LIN {X 0,Y 409.894,Z 382.469,A -85,B 0,C 180,E1 -10359.873,E2 -10359.873} C_VEL
LIN {X 0,Y 410.199,Z 379.368,A -85,B 0,C 180,E1 -10361.865,E2 -10361.865} C_VEL
LIN {X 0,Y 410.49,Z 374.761,A -85,B 0,C 180,E1 -10363.869,E2 -10363.869} C_VEL
LIN {X 0,Y 410.864,Z 370.201,A -85,B 0,C 180,E1 -10365.375,E2 -10365.375} C_VEL
LIN {X 0,Y 411.455,Z 364.311,A -85,B 0,C 180,E1 -10366.955,E2 -10366.955} C_VEL
LIN {X 0,Y 412.195,Z 356.607,A -85,B 0,C 180,E1 -10368.644,E2 -10368.644} C_VEL
LIN {X 0,Y 413.203,Z 347.062,A -85,B 0,C 180,E1 -10370.341,E2 -10370.341} C_VEL
LIN {X 0,Y 414.197,Z 338.033,A -85,B 0,C 180,E1 -10371.657,E2 -10371.657} C_VEL
LIN {X 0,Y 415.184,Z 327.747,A -85,B 0,C 180,E1 -10372.913,E2 -10372.913} C_VEL
LIN {X 0,Y 416.321,Z 316.334,A -85,B 0,C 180,E1 -10374.056,E2 -10374.056} C_VEL
LIN {X 0,Y 417.327,Z 304.389,A -85,B 0,C 180,E1 -10375.032,E2 -10375.032} C_VEL
LIN {X 0,Y 418.436,Z 290.839,A -85,B 0,C 180,E1 -10375.893,E2 -10375.893} C_VEL
LIN {X 0,Y 419.174,Z 276.579,A -85,B 0,C 180,E1 -10376.58,E2 -10376.58} C_VEL
LIN {X 0,Y 419.797,Z 262.212,A -85,B 0,C 180,E1 -10377.052,E2 -10377.052} C_VEL
LIN {X 0,Y 420.231,Z 239.052,A -85,B 0,C 180,E1 -10377.499,E2 -10377.499} C_VEL
LIN {X 0,Y 421.741,Z 148.538,A -85,B 0,C 180,E1 -10379.069,E2 -10379.069} C_VEL
LIN {X 0,Y 417.255,Z 129.702,A -85,B 0,C 180,E1 -10379.713,E2 -10379.713} C_VEL
LIN {X 0,Y 414.712,Z 123.273,A -85,B 0,C 180,E1 -10380.021,E2 -10380.021} C_VEL
LIN {X 0,Y 411.925,Z 110.451,A -85,B 0,C 180,E1 -10383.091,E2 -10383.091} C_VEL
LIN {X 0,Y 411.225,Z 107.391,A -85,B 0,C 180,E1 -10383.888,E2 -10383.888} C_VEL
LIN {X 0,Y 411.186,Z 107.387,A -85,B 0,C 180,E1 -10386.743,E2 -10386.743} C_VEL
LIN {X 0,Y 411.164,Z 107.396,A -85,B 0,C 180,E1 -10389.719,E2 -10389.719} C_VEL
LIN {X 0,Y 411.162,Z 107.393,A -85,B 0,C 180,E1 -10393.135,E2 -10393.135} C_VEL
LIN {X 0,Y 411.164,Z 107.386,A -85,B 0,C 180,E1 -10395.882,E2 -10395.882} C_VEL
LIN {X 0,Y 411.148,Z 107.394,A -85,B 0,C 180,E1 -10398.774,E2 -10398.774} C_VEL
LIN {X 0,Y 411.183,Z 107.39,A -85,B 0,C 180,E1 -10402.025,E2 -10402.025} C_VEL
LIN {X 0,Y 411.203,Z 107.389,A -85,B 0,C 180,E1 -10405.123,E2 -10405.123} C_VEL
LIN {X 0,Y 411.166,Z 107.391,A -85,B 0,C 180,E1 -10408.002,E2 -10408.002} C_VEL
LIN {X 0,Y 411.181,Z 107.392,A -85,B 0,C 180,E1 -10411.407,E2 -10411.407} C_VEL
LIN {X 0,Y 411.213,Z 107.388,A -85,B 0,C 180,E1 -10414.934,E2 -10414.934} C_VEL
LIN {X 0,Y 411.204,Z 107.38,A -85,B 0,C 180,E1 -10417.913,E2 -10417.913} C_VEL
LIN {X 0,Y 411.22,Z 107.381,A -85,B 0,C 180,E1 -10421.051,E2 -10421.051} C_VEL
LIN {X 0,Y 411.254,Z 107.382,A -85,B 0,C 180,E1 -10424.131,E2 -10424.131} C_VEL
LIN {X 0,Y 411.304,Z 107.371,A -85,B 0,C 180,E1 -10427.165,E2 -10427.165} C_VEL
LIN {X 0,Y 411.292,Z 107.375,A -85,B 0,C 180,E1 -10430.161,E2 -10430.161} C_VEL
LIN {X 0,Y 411.424,Z 107.358,A -85,B 0,C 180,E1 -10433.132,E2 -10433.132} C_VEL
LIN {X 0,Y 411.304,Z 107.371,A -85,B 0,C 180,E1 -10435.099,E2 -10435.099} C_VEL
LIN {X 0,Y 411.511,Z 107.351,A -85,B 0,C 180,E1 -10438.042,E2 -10438.042} C_VEL
LIN {X 0,Y 411.639,Z 107.332,A -85,B 0,C 180,E1 -10440,E2 -10440} C_VEL
LIN {X 0,Y 411.451,Z 107.354,A -85,B 0,C 180,E1 -10442.937,E2 -10442.937} C_VEL
LIN {X 0,Y 411.435,Z 107.353,A -85,B 0,C 180,E1 -10445.882,E2 -10445.882} C_VEL
LIN {X 0,Y 411.319,Z 107.372,A -85,B 0,C 180,E1 -10448.846,E2 -10448.846} C_VEL
LIN {X 0,Y 411.284,Z 107.374,A -85,B 0,C 180,E1 -10451.833,E2 -10451.833} C_VEL
LIN {X 0,Y 411.26,Z 107.38,A -85,B 0,C 180,E1 -10454.853,E2 -10454.853} C_VEL
LIN {X 0,Y 411.253,Z 107.38,A -85,B 0,C 180,E1 -10457.915,E2 -10457.915} C_VEL
LIN {X 0,Y 411.197,Z 107.383,A -85,B 0,C 180,E1 -10461.034,E2 -10461.034} C_VEL
LIN {X 0,Y 411.228,Z 107.38,A -85,B 0,C 180,E1 -10464.215,E2 -10464.215} C_VEL
LIN {X 0,Y 411.259,Z 107.378,A -85,B 0,C 180,E1 -10467.478,E2 -10467.478} C_VEL
LIN {X 0,Y 411.19,Z 107.392,A -85,B 0,C 180,E1 -10470.847,E2 -10470.847} C_VEL
LIN {X 0,Y 411.207,Z 107.389,A -85,B 0,C 180,E1 -10474.333,E2 -10474.333} C_VEL
LIN {X 0,Y 411.192,Z 107.389,A -85,B 0,C 180,E1 -10477.974,E2 -10477.974} C_VEL
LIN {X 0,Y 411.164,Z 107.39,A -85,B 0,C 180,E1 -10481.228,E2 -10481.228} C_VEL
LIN {X 0,Y 411.176,Z 107.383,A -85,B 0,C 180,E1 -10484.49,E2 -10484.49} C_VEL
LIN {X 0,Y 411.178,Z 107.394,A -85,B 0,C 180,E1 -10488.195,E2 -10488.195} C_VEL
LIN {X 0,Y 411.223,Z 107.382,A -85,B 0,C 180,E1 -10490.776,E2 -10490.776} C_VEL
LIN {X 0,Y 411.199,Z 107.386,A -85,B 0,C 180,E1 -10494.471,E2 -10494.471} C_VEL
LIN {X 0,Y 411.208,Z 107.379,A -85,B 0,C 180,E1 -10496.873,E2 -10496.873} C_VEL
LIN {X 0,Y 411.225,Z 107.421,A -85,B 0,C 180,E1 -10499.227,E2 -10499.227} C_VEL
LIN {X 0,Y 414.619,Z 121.415,A -85,B 0,C 180,E1 -10502.366,E2 -10502.366} C_VEL
LIN {X 0,Y 416.242,Z 130.214,A -85,B 0,C 180,E1 -10504.229,E2 -10504.229} C_VEL
LIN {X 0,Y 415.402,Z 139.95,A -85,B 0,C 180,E1 -10506.075,E2 -10506.075} C_VEL
LIN {X 0,Y 421.021,Z 167.755,A -85,B 0,C 180,E1 -10506.967,E2 -10506.967} C_VEL
LIN {X 0,Y 421.464,Z 172.933,A -85,B 0,C 180,E1 -10507.09,E2 -10507.09} C_VEL
LIN {X 0,Y 419.669,Z 277.802,A -85,B 0,C 180,E1 -10508.929,E2 -10508.929} C_VEL
LIN {X 0,Y 418.967,Z 292.415,A -85,B 0,C 180,E1 -10509.374,E2 -10509.374} C_VEL
LIN {X 0,Y 418.091,Z 305.794,A -85,B 0,C 180,E1 -10509.971,E2 -10509.971} C_VEL
LIN {X 0,Y 417.093,Z 319.845,A -85,B 0,C 180,E1 -10510.825,E2 -10510.825} C_VEL
LIN {X 0,Y 416.008,Z 332.243,A -85,B 0,C 180,E1 -10511.788,E2 -10511.788} C_VEL
LIN {X 0,Y 414.859,Z 343.663,A -85,B 0,C 180,E1 -10512.882,E2 -10512.882} C_VEL
LIN {X 0,Y 413.673,Z 355.136,A -85,B 0,C 180,E1 -10514.227,E2 -10514.227} C_VEL
LIN {X 0,Y 412.634,Z 365.412,A -85,B 0,C 180,E1 -10515.702,E2 -10515.702} C_VEL
LIN {X 0,Y 411.827,Z 373.917,A -85,B 0,C 180,E1 -10517.182,E2 -10517.182} C_VEL
LIN {X 0,Y 411.039,Z 382.063,A -85,B 0,C 180,E1 -10518.91,E2 -10518.91} C_VEL
LIN {X 0,Y 410.52,Z 388.644,A -85,B 0,C 180,E1 -10520.64,E2 -10520.64} C_VEL
LIN {X 0,Y 410.161,Z 394.498,A -85,B 0,C 180,E1 -10522.616,E2 -10522.616} C_VEL
LIN {X 0,Y 409.998,Z 397.888,A -85,B 0,C 180,E1 -10524.097,E2 -10524.097} C_VEL
LIN {X 0,Y 409.904,Z 401.081,A -85,B 0,C 180,E1 -10526.067,E2 -10526.067} C_VEL
LIN {X 0,Y 409.958,Z 402.906,A -85,B 0,C 180,E1 -10528.035,E2 -10528.035} C_VEL
LIN {X 0,Y 409.905,Z 403.396,A -85,B 0,C 180,E1 -10530,E2 -10530} C_VEL
LIN {X 0,Y 409.963,Z 402.557,A -85,B 0,C 180,E1 -10531.965,E2 -10531.965} C_VEL
LIN {X 0,Y 409.904,Z 400.363,A -85,B 0,C 180,E1 -10533.932,E2 -10533.932} C_VEL
LIN {X 0,Y 409.976,Z 396.757,A -85,B 0,C 180,E1 -10535.903,E2 -10535.903} C_VEL
LIN {X 0,Y 410.181,Z 391.629,A -85,B 0,C 180,E1 -10537.878,E2 -10537.878} C_VEL
LIN {X 0,Y 410.447,Z 386.655,A -85,B 0,C 180,E1 -10539.362,E2 -10539.362} C_VEL
LIN {X 0,Y 410.935,Z 379.509,A -85,B 0,C 180,E1 -10541.093,E2 -10541.093} C_VEL
LIN {X 0,Y 411.493,Z 372.023,A -85,B 0,C 180,E1 -10542.577,E2 -10542.577} C_VEL
LIN {X 0,Y 412.153,Z 363.017,A -85,B 0,C 180,E1 -10544.063,E2 -10544.063} C_VEL
LIN {X 0,Y 412.956,Z 354.075,A -85,B 0,C 180,E1 -10545.295,E2 -10545.295} C_VEL
LIN {X 0,Y 413.778,Z 343.393,A -85,B 0,C 180,E1 -10546.529,E2 -10546.529} C_VEL
LIN {X 0,Y 414.78,Z 331.746,A -85,B 0,C 180,E1 -10547.63,E2 -10547.63} C_VEL
LIN {X 0,Y 415.787,Z 318.934,A -85,B 0,C 180,E1 -10548.605,E2 -10548.605} C_VEL
LIN {X 0,Y 416.63,Z 305.594,A -85,B 0,C 180,E1 -10549.399,E2 -10549.399} C_VEL
LIN {X 0,Y 417.339,Z 291.973,A -85,B 0,C 180,E1 -10550.002,E2 -10550.002} C_VEL
LIN {X 0,Y 417.882,Z 278.039,A -85,B 0,C 180,E1 -10550.425,E2 -10550.425} C_VEL
LIN {X 0,Y 419.494,Z 169.965,A -85,B 0,C 180,E1 -10552.298,E2 -10552.298} C_VEL
LIN {X 0,Y 414.351,Z 140.071,A -85,B 0,C 180,E1 -10553.116,E2 -10553.116} C_VEL
LIN {X 0,Y 415.279,Z 126.829,A -85,B 0,C 180,E1 -10555.566,E2 -10555.566} C_VEL
LIN {X 0,Y 413.122,Z 115.869,A -85,B 0,C 180,E1 -10557.795,E2 -10557.795} C_VEL
LIN {X 0,Y 411.225,Z 107.388,A -85,B 0,C 180,E1 -10559.597,E2 -10559.597} C_VEL
LIN {X 0,Y 411.206,Z 107.385,A -85,B 0,C 180,E1 -10563.156,E2 -10563.156} C_VEL
LIN {X 0,Y 411.192,Z 107.388,A -85,B 0,C 180,E1 -10566.552,E2 -10566.552} C_VEL
LIN {X 0,Y 411.212,Z 107.388,A -85,B 0,C 180,E1 -10569.728,E2 -10569.728} C_VEL
LIN {X 0,Y 411.174,Z 107.389,A -85,B 0,C 180,E1 -10573.133,E2 -10573.133} C_VEL
LIN {X 0,Y 411.233,Z 107.387,A -85,B 0,C 180,E1 -10575.871,E2 -10575.871} C_VEL
LIN {X 0,Y 411.204,Z 107.385,A -85,B 0,C 180,E1 -10578.765,E2 -10578.765} C_VEL
LIN {X 0,Y 411.19,Z 107.389,A -85,B 0,C 180,E1 -10582.026,E2 -10582.026} C_VEL
LIN {X 0,Y 411.204,Z 107.389,A -85,B 0,C 180,E1 -10585.666,E2 -10585.666} C_VEL
LIN {X 0,Y 411.188,Z 107.392,A -85,B 0,C 180,E1 -10589.152,E2 -10589.152} C_VEL
LIN {X 0,Y 411.257,Z 107.379,A -85,B 0,C 180,E1 -10592.522,E2 -10592.522} C_VEL
LIN {X 0,Y 411.225,Z 107.383,A -85,B 0,C 180,E1 -10595.785,E2 -10595.785} C_VEL
LIN {X 0,Y 411.195,Z 107.393,A -85,B 0,C 180,E1 -10598.966,E2 -10598.966} C_VEL
LIN {X 0,Y 411.251,Z 107.379,A -85,B 0,C 180,E1 -10602.085,E2 -10602.085} C_VEL
LIN {X 0,Y 411.259,Z 107.381,A -85,B 0,C 180,E1 -10605.147,E2 -10605.147} C_VEL
LIN {X 0,Y 411.283,Z 107.377,A -85,B 0,C 180,E1 -10608.167,E2 -10608.167} C_VEL
LIN {X 0,Y 411.439,Z 107.358,A -85,B 0,C 180,E1 -10612.189,E2 -10612.189} C_VEL
LIN {X 0,Y 411.471,Z 107.354,A -85,B 0,C 180,E1 -10614.118,E2 -10614.118} C_VEL
LIN {X 0,Y 411.51,Z 107.35,A -85,B 0,C 180,E1 -10618.043,E2 -10618.043} C_VEL
LIN {X 0,Y 411.639,Z 107.334,A -85,B 0,C 180,E1 -10620,E2 -10620} C_VEL
LIN {X 0,Y 411.457,Z 107.354,A -85,B 0,C 180,E1 -10622.937,E2 -10622.937} C_VEL
LIN {X 0,Y 411.421,Z 107.358,A -85,B 0,C 180,E1 -10626.528,E2 -10626.528} C_VEL
LIN {X 0,Y 411.292,Z 107.379,A -85,B 0,C 180,E1 -10629.839,E2 -10629.839} C_VEL
LIN {X 0,Y 411.305,Z 107.373,A -85,B 0,C 180,E1 -10633.104,E2 -10633.104} C_VEL
LIN {X 0,Y 411.257,Z 107.378,A -85,B 0,C 180,E1 -10636.889,E2 -10636.889} C_VEL
LIN {X 0,Y 411.23,Z 107.385,A -85,B 0,C 180,E1 -10639.987,E2 -10639.987} C_VEL
LIN {X 0,Y 411.202,Z 107.388,A -85,B 0,C 180,E1 -10643.148,E2 -10643.148} C_VEL
LIN {X 0,Y 411.236,Z 107.381,A -85,B 0,C 180,E1 -10646.381,E2 -10646.381} C_VEL
LIN {X 0,Y 411.2,Z 107.388,A -85,B 0,C 180,E1 -10649.713,E2 -10649.713} C_VEL
LIN {X 0,Y 411.206,Z 107.391,A -85,B 0,C 180,E1 -10653.156,E2 -10653.156} C_VEL
LIN {X 0,Y 411.192,Z 107.388,A -85,B 0,C 180,E1 -10656.553,E2 -10656.553} C_VEL
LIN {X 0,Y 411.209,Z 107.385,A -85,B 0,C 180,E1 -10659.728,E2 -10659.728} C_VEL
LIN {X 0,Y 411.173,Z 107.393,A -85,B 0,C 180,E1 -10663.134,E2 -10663.134} C_VEL
LIN {X 0,Y 411.168,Z 107.389,A -85,B 0,C 180,E1 -10665.882,E2 -10665.882} C_VEL
LIN {X 0,Y 411.161,Z 107.396,A -85,B 0,C 180,E1 -10668.773,E2 -10668.773} C_VEL
LIN {X 0,Y 411.19,Z 107.388,A -85,B 0,C 180,E1 -10672.026,E2 -10672.026} C_VEL
LIN {X 0,Y 411.207,Z 107.385,A -85,B 0,C 180,E1 -10675.667,E2 -10675.667} C_VEL
LIN {X 0,Y 411.19,Z 107.387,A -85,B 0,C 180,E1 -10679.153,E2 -10679.153} C_VEL
LIN {X 0,Y 411.19,Z 107.39,A -85,B 0,C 180,E1 -10682.518,E2 -10682.518} C_VEL
LIN {X 0,Y 411.213,Z 107.387,A -85,B 0,C 180,E1 -10685.784,E2 -10685.784} C_VEL
LIN {X 0,Y 411.265,Z 107.528,A -85,B 0,C 180,E1 -10689.428,E2 -10689.428} C_VEL
LIN {X 0,Y 413.796,Z 119.688,A -85,B 0,C 180,E1 -10692.199,E2 -10692.199} C_VEL
LIN {X 0,Y 414.458,Z 123.421,A -85,B 0,C 180,E1 -10692.975,E2 -10692.975} C_VEL
LIN {X 0,Y 417.105,Z 135.031,A -85,B 0,C 180,E1 -10693.325,E2 -10693.325} C_VEL
LIN {X 0,Y 419.723,Z 149.234,A -85,B 0,C 180,E1 -10693.716,E2 -10693.716} C_VEL
LIN {X 0,Y 418.093,Z 260.183,A -85,B 0,C 180,E1 -10695.644,E2 -10695.644} C_VEL
LIN {X 0,Y 417.665,Z 274.581,A -85,B 0,C 180,E1 -10696.095,E2 -10696.095} C_VEL
LIN {X 0,Y 416.965,Z 288.413,A -85,B 0,C 180,E1 -10696.724,E2 -10696.724} C_VEL
LIN {X 0,Y 416.084,Z 302.171,A -85,B 0,C 180,E1 -10697.564,E2 -10697.564} C_VEL
LIN {X 0,Y 415.231,Z 314.486,A -85,B 0,C 180,E1 -10698.529,E2 -10698.529} C_VEL
LIN {X 0,Y 414.251,Z 326.918,A -85,B 0,C 180,E1 -10699.739,E2 -10699.739} C_VEL
LIN {X 0,Y 413.54,Z 335.173,A -85,B 0,C 180,E1 -10700.711,E2 -10700.711} C_VEL
LIN {X 0,Y 412.551,Z 339.509,A -85,B 0,C 180,E1 -10701.255,E2 -10701.255} C_VEL
LIN {X 0,Y 409.156,Z 346.272,A -85,B 0,C 180,E1 -10702.152,E2 -10702.152} C_VEL
LIN {X 0,Y 405.739,Z 352.574,A -85,B 0,C 180,E1 -10703.119,E2 -10703.119} C_VEL
LIN {X 0,Y 404.726,Z 356.126,A -85,B 0,C 180,E1 -10703.766,E2 -10703.766} C_VEL
LIN {X 0,Y 403.983,Z 364.113,A -85,B 0,C 180,E1 -10705.51,E2 -10705.51} C_VEL
LIN {X 0,Y 403.476,Z 369.74,A -85,B 0,C 180,E1 -10707.005,E2 -10707.005} C_VEL
LIN {X 0,Y 403.107,Z 375.638,A -85,B 0,C 180,E1 -10709.001,E2 -10709.001} C_VEL
LIN {X 0,Y 402.938,Z 379.979,A -85,B 0,C 180,E1 -10711,E2 -10711} C_VEL
LIN {X 0,Y 402.855,Z 382.89,A -85,B 0,C 180,E1 -10713,E2 -10713} C_VEL
LIN {X 0,Y 402.857,Z 384.45,A -85,B 0,C 180,E1 -10715.004,E2 -10715.004} C_VEL
LIN {X 0,Y 402.849,Z 384.69,A -85,B 0,C 180,E1 -10717.015,E2 -10717.015} C_VEL
LIN {X 0,Y 402.79,Z 383.602,A -85,B 0,C 180,E1 -10719.035,E2 -10719.035} C_VEL
LIN {X 0,Y 403.005,Z 381.155,A -85,B 0,C 180,E1 -10721.06,E2 -10721.06} C_VEL
LIN {X 0,Y 403.282,Z 377.264,A -85,B 0,C 180,E1 -10723.094,E2 -10723.094} C_VEL
LIN {X 0,Y 403.718,Z 371.756,A -85,B 0,C 180,E1 -10725.137,E2 -10725.137} C_VEL
LIN {X 0,Y 404.458,Z 364.731,A -85,B 0,C 180,E1 -10727.117,E2 -10727.117} C_VEL
LIN {X 0,Y 405.173,Z 357.658,A -85,B 0,C 180,E1 -10728.717,E2 -10728.717} C_VEL
LIN {X 0,Y 406.244,Z 348.306,A -85,B 0,C 180,E1 -10730.442,E2 -10730.442} C_VEL
LIN {X 0,Y 407.248,Z 339.488,A -85,B 0,C 180,E1 -10731.779,E2 -10731.779} C_VEL
LIN {X 0,Y 408.267,Z 329.465,A -85,B 0,C 180,E1 -10733.056,E2 -10733.056} C_VEL
LIN {X 0,Y 409.405,Z 318.622,A -85,B 0,C 180,E1 -10734.195,E2 -10734.195} C_VEL
LIN {X 0,Y 410.498,Z 306.717,A -85,B 0,C 180,E1 -10735.221,E2 -10735.221} C_VEL
LIN {X 0,Y 411.711,Z 293.073,A -85,B 0,C 180,E1 -10736.144,E2 -10736.144} C_VEL
LIN {X 0,Y 412.504,Z 279.641,A -85,B 0,C 180,E1 -10736.84,E2 -10736.84} C_VEL
LIN {X 0,Y 413.151,Z 265.955,A -85,B 0,C 180,E1 -10737.341,E2 -10737.341} C_VEL
LIN {X 0,Y 413.591,Z 250.535,A -85,B 0,C 180,E1 -10737.689,E2 -10737.689} C_VEL
LIN {X 0,Y 415.285,Z 149.52,A -85,B 0,C 180,E1 -10739.472,E2 -10739.472} C_VEL
LIN {X 0,Y 411.167,Z 132.309,A -85,B 0,C 180,E1 -10740.077,E2 -10740.077} C_VEL
LIN {X 0,Y 407.563,Z 123.457,A -85,B 0,C 180,E1 -10740.515,E2 -10740.515} C_VEL
LIN {X 0,Y 405.275,Z 112.902,A -85,B 0,C 180,E1 -10743.087,E2 -10743.087} C_VEL
LIN {X 0,Y 404.156,Z 108.267,A -85,B 0,C 180,E1 -10744.262,E2 -10744.262} C_VEL
LIN {X 0,Y 404.132,Z 108.267,A -85,B 0,C 180,E1 -10747.493,E2 -10747.493} C_VEL
LIN {X 0,Y 404.118,Z 108.273,A -85,B 0,C 180,E1 -10750.075,E2 -10750.075} C_VEL
LIN {X 0,Y 404.142,Z 108.268,A -85,B 0,C 180,E1 -10753.082,E2 -10753.082} C_VEL
LIN {X 0,Y 404.121,Z 108.263,A -85,B 0,C 180,E1 -10755.922,E2 -10755.922} C_VEL
LIN {X 0,Y 404.103,Z 108.272,A -85,B 0,C 180,E1 -10758.632,E2 -10758.632} C_VEL
LIN {X 0,Y 404.139,Z 108.264,A -85,B 0,C 180,E1 -10761.495,E2 -10761.495} C_VEL
LIN {X 0,Y 404.174,Z 108.263,A -85,B 0,C 180,E1 -10764.983,E2 -10764.983} C_VEL
LIN {X 0,Y 404.14,Z 108.267,A -85,B 0,C 180,E1 -10768.442,E2 -10768.442} C_VEL
LIN {X 0,Y 404.153,Z 108.264,A -85,B 0,C 180,E1 -10770.862,E2 -10770.862} C_VEL
LIN {X 0,Y 404.141,Z 108.262,A -85,B 0,C 180,E1 -10774.23,E2 -10774.23} C_VEL
LIN {X 0,Y 404.167,Z 108.257,A -85,B 0,C 180,E1 -10777.508,E2 -10777.508} C_VEL
LIN {X 0,Y 404.163,Z 108.264,A -85,B 0,C 180,E1 -10780.707,E2 -10780.707} C_VEL
LIN {X 0,Y 404.222,Z 108.256,A -85,B 0,C 180,E1 -10783.848,E2 -10783.848} C_VEL
LIN {X 0,Y 404.284,Z 108.247,A -85,B 0,C 180,E1 -10786.939,E2 -10786.939} C_VEL
LIN {X 0,Y 404.257,Z 108.254,A -85,B 0,C 180,E1 -10789.988,E2 -10789.988} C_VEL
LIN {X 0,Y 404.37,Z 108.237,A -85,B 0,C 180,E1 -10793.012,E2 -10793.012} C_VEL
LIN {X 0,Y 404.276,Z 108.246,A -85,B 0,C 180,E1 -10795.013,E2 -10795.013} C_VEL
LIN {X 0,Y 404.479,Z 108.227,A -85,B 0,C 180,E1 -10798.008,E2 -10798.008} C_VEL
LIN {X 0,Y 404.608,Z 108.207,A -85,B 0,C 180,E1 -10800,E2 -10800} C_VEL
LIN {X 0,Y 404.409,Z 108.231,A -85,B 0,C 180,E1 -10802.988,E2 -10802.988} C_VEL
LIN {X 0,Y 404.382,Z 108.23,A -85,B 0,C 180,E1 -10805.985,E2 -10805.985} C_VEL
LIN {X 0,Y 404.266,Z 108.251,A -85,B 0,C 180,E1 -10809.001,E2 -10809.001} C_VEL
LIN {X 0,Y 404.256,Z 108.25,A -85,B 0,C 180,E1 -10812.041,E2 -10812.041} C_VEL
LIN {X 0,Y 404.207,Z 108.259,A -85,B 0,C 180,E1 -10815.118,E2 -10815.118} C_VEL
LIN {X 0,Y 404.211,Z 108.256,A -85,B 0,C 180,E1 -10818.238,E2 -10818.238} C_VEL
LIN {X 0,Y 404.139,Z 108.264,A -85,B 0,C 180,E1 -10821.419,E2 -10821.419} C_VEL
LIN {X 0,Y 404.178,Z 108.259,A -85,B 0,C 180,E1 -10824.665,E2 -10824.665} C_VEL
LIN {X 0,Y 404.196,Z 108.257,A -85,B 0,C 180,E1 -10827.999,E2 -10827.999} C_VEL
LIN {X 0,Y 404.14,Z 108.264,A -85,B 0,C 180,E1 -10831.558,E2 -10831.558} C_VEL
LIN {X 0,Y 404.185,Z 108.259,A -85,B 0,C 180,E1 -10835.016,E2 -10835.016} C_VEL
LIN {X 0,Y 404.151,Z 108.257,A -85,B 0,C 180,E1 -10838.757,E2 -10838.757} C_VEL
LIN {X 0,Y 404.123,Z 108.267,A -85,B 0,C 180,E1 -10841.6,E2 -10841.6} C_VEL
LIN {X 0,Y 404.146,Z 108.258,A -85,B 0,C 180,E1 -10844.522,E2 -10844.522} C_VEL
LIN {X 0,Y 404.137,Z 108.267,A -85,B 0,C 180,E1 -10847.296,E2 -10847.296} C_VEL
LIN {X 0,Y 404.169,Z 108.265,A -85,B 0,C 180,E1 -10849.955,E2 -10849.955} C_VEL
LIN {X 0,Y 404.137,Z 108.265,A -85,B 0,C 180,E1 -10853.125,E2 -10853.125} C_VEL
LIN {X 0,Y 404.146,Z 108.263,A -85,B 0,C 180,E1 -10856.188,E2 -10856.188} C_VEL
LIN {X 0,Y 404.155,Z 108.364,A -85,B 0,C 180,E1 -10858.81,E2 -10858.81} C_VEL
LIN {X 0,Y 407.451,Z 121.693,A -85,B 0,C 180,E1 -10861.878,E2 -10861.878} C_VEL
LIN {X 0,Y 409.264,Z 130.276,A -85,B 0,C 180,E1 -10863.756,E2 -10863.756} C_VEL
LIN {X 0,Y 409.21,Z 134.367,A -85,B 0,C 180,E1 -10864.573,E2 -10864.573} C_VEL
LIN {X 0,Y 408.716,Z 139.926,A -85,B 0,C 180,E1 -10865.626,E2 -10865.626} C_VEL
LIN {X 0,Y 414.416,Z 167.889,A -85,B 0,C 180,E1 -10866.544,E2 -10866.544} C_VEL
LIN {X 0,Y 415.022,Z 173.117,A -85,B 0,C 180,E1 -10866.682,E2 -10866.682} C_VEL
LIN {X 0,Y 413.145,Z 277.83,A -85,B 0,C 180,E1 -10868.547,E2 -10868.547} C_VEL
LIN {X 0,Y 412.398,Z 292.374,A -85,B 0,C 180,E1 -10868.997,E2 -10868.997} C_VEL
LIN {X 0,Y 411.444,Z 306.283,A -85,B 0,C 180,E1 -10869.633,E2 -10869.633} C_VEL
LIN {X 0,Y 410.398,Z 320.192,A -85,B 0,C 180,E1 -10870.499,E2 -10870.499} C_VEL
LIN {X 0,Y 409.272,Z 332.489,A -85,B 0,C 180,E1 -10871.477,E2 -10871.477} C_VEL
LIN {X 0,Y 408.079,Z 343.835,A -85,B 0,C 180,E1 -10872.588,E2 -10872.588} C_VEL
LIN {X 0,Y 406.82,Z 355.25,A -85,B 0,C 180,E1 -10873.954,E2 -10873.954} C_VEL
LIN {X 0,Y 405.708,Z 365.463,A -85,B 0,C 180,E1 -10875.452,E2 -10875.452} C_VEL
LIN {X 0,Y 404.84,Z 373.934,A -85,B 0,C 180,E1 -10876.957,E2 -10876.957} C_VEL
LIN {X 0,Y 404.043,Z 382.04,A -85,B 0,C 180,E1 -10878.715,E2 -10878.715} C_VEL
LIN {X 0,Y 403.497,Z 388.592,A -85,B 0,C 180,E1 -10880.475,E2 -10880.475} C_VEL
LIN {X 0,Y 403.089,Z 394.419,A -85,B 0,C 180,E1 -10882.486,E2 -10882.486} C_VEL
LIN {X 0,Y 402.937,Z 397.788,A -85,B 0,C 180,E1 -10883.993,E2 -10883.993} C_VEL
LIN {X 0,Y 402.825,Z 400.956,A -85,B 0,C 180,E1 -10885.998,E2 -10885.998} C_VEL
LIN {X 0,Y 402.854,Z 402.759,A -85,B 0,C 180,E1 -10888,E2 -10888} C_VEL
LIN {X 0,Y 402.831,Z 403.228,A -85,B 0,C 180,E1 -10890,E2 -10890} C_VEL
LIN {X 0,Y 402.86,Z 402.367,A -85,B 0,C 180,E1 -10891.999,E2 -10891.999} C_VEL
LIN {X 0,Y 402.824,Z 400.151,A -85,B 0,C 180,E1 -10894.002,E2 -10894.002} C_VEL
LIN {X 0,Y 402.897,Z 396.521,A -85,B 0,C 180,E1 -10896.008,E2 -10896.008} C_VEL
LIN {X 0,Y 403.126,Z 391.368,A -85,B 0,C 180,E1 -10898.017,E2 -10898.017} C_VEL
LIN {X 0,Y 403.382,Z 386.366,A -85,B 0,C 180,E1 -10899.527,E2 -10899.527} C_VEL
LIN {X 0,Y 403.924,Z 379.191,A -85,B 0,C 180,E1 -10901.288,E2 -10901.288} C_VEL
LIN {X 0,Y 404.625,Z 370.302,A -85,B 0,C 180,E1 -10903.05,E2 -10903.05} C_VEL
LIN {X 0,Y 405.325,Z 360.979,A -85,B 0,C 180,E1 -10904.561,E2 -10904.561} C_VEL
LIN {X 0,Y 406.255,Z 350.664,A -85,B 0,C 180,E1 -10905.94,E2 -10905.94} C_VEL
LIN {X 0,Y 407.337,Z 339.288,A -85,B 0,C 180,E1 -10907.185,E2 -10907.185} C_VEL
LIN {X 0,Y 408.239,Z 328.276,A -85,B 0,C 180,E1 -10908.181,E2 -10908.181} C_VEL
LIN {X 0,Y 409.215,Z 315.314,A -85,B 0,C 180,E1 -10909.121,E2 -10909.121} C_VEL
LIN {X 0,Y 410.073,Z 301.3,A -85,B 0,C 180,E1 -10909.902,E2 -10909.902} C_VEL
LIN {X 0,Y 410.802,Z 287.272,A -85,B 0,C 180,E1 -10910.465,E2 -10910.465} C_VEL
LIN {X 0,Y 411.275,Z 273.236,A -85,B 0,C 180,E1 -10910.833,E2 -10910.833} C_VEL
LIN {X 0,Y 412.779,Z 170.459,A -85,B 0,C 180,E1 -10912.63,E2 -10912.63} C_VEL
LIN {X 0,Y 407.545,Z 139.875,A -85,B 0,C 180,E1 -10913.491,E2 -10913.491} C_VEL
LIN {X 0,Y 408.359,Z 128.088,A -85,B 0,C 180,E1 -10915.714,E2 -10915.714} C_VEL
LIN {X 0,Y 406.107,Z 116.868,A -85,B 0,C 180,E1 -10918.043,E2 -10918.043} C_VEL
LIN {X 0,Y 404.189,Z 108.264,A -85,B 0,C 180,E1 -10919.899,E2 -10919.899} C_VEL
LIN {X 0,Y 404.145,Z 108.267,A -85,B 0,C 180,E1 -10923.812,E2 -10923.812} C_VEL
LIN {X 0,Y 404.136,Z 108.266,A -85,B 0,C 180,E1 -10926.875,E2 -10926.875} C_VEL
LIN {X 0,Y 404.146,Z 108.27,A -85,B 0,C 180,E1 -10930.08,E2 -10930.08} C_VEL
LIN {X 0,Y 404.153,Z 108.264,A -85,B 0,C 180,E1 -10933.084,E2 -10933.084} C_VEL
LIN {X 0,Y 404.206,Z 108.262,A -85,B 0,C 180,E1 -10935.934,E2 -10935.934} C_VEL
LIN {X 0,Y 404.159,Z 108.262,A -85,B 0,C 180,E1 -10938.64,E2 -10938.64} C_VEL
LIN {X 0,Y 404.149,Z 108.27,A -85,B 0,C 180,E1 -10941.493,E2 -10941.493} C_VEL
LIN {X 0,Y 404.183,Z 108.261,A -85,B 0,C 180,E1 -10944.984,E2 -10944.984} C_VEL
LIN {X 0,Y 404.14,Z 108.265,A -85,B 0,C 180,E1 -10948.554,E2 -10948.554} C_VEL
LIN {X 0,Y 404.194,Z 108.258,A -85,B 0,C 180,E1 -10952,E2 -10952} C_VEL
LIN {X 0,Y 404.176,Z 108.265,A -85,B 0,C 180,E1 -10955.334,E2 -10955.334} C_VEL
LIN {X 0,Y 404.137,Z 108.267,A -85,B 0,C 180,E1 -10958.581,E2 -10958.581} C_VEL
LIN {X 0,Y 404.209,Z 108.256,A -85,B 0,C 180,E1 -10961.762,E2 -10961.762} C_VEL
LIN {X 0,Y 404.205,Z 108.263,A -85,B 0,C 180,E1 -10964.882,E2 -10964.882} C_VEL
LIN {X 0,Y 404.255,Z 108.251,A -85,B 0,C 180,E1 -10967.959,E2 -10967.959} C_VEL
LIN {X 0,Y 404.404,Z 108.234,A -85,B 0,C 180,E1 -10972.129,E2 -10972.129} C_VEL
LIN {X 0,Y 404.419,Z 108.232,A -85,B 0,C 180,E1 -10974.015,E2 -10974.015} C_VEL
LIN {X 0,Y 404.479,Z 108.225,A -85,B 0,C 180,E1 -10978.009,E2 -10978.009} C_VEL
LIN {X 0,Y 404.608,Z 108.21,A -85,B 0,C 180,E1 -10980,E2 -10980} C_VEL
LIN {X 0,Y 404.415,Z 108.231,A -85,B 0,C 180,E1 -10982.989,E2 -10982.989} C_VEL
LIN {X 0,Y 404.37,Z 108.237,A -85,B 0,C 180,E1 -10986.524,E2 -10986.524} C_VEL
LIN {X 0,Y 404.288,Z 108.246,A -85,B 0,C 180,E1 -10989.001,E2 -10989.001} C_VEL
LIN {X 0,Y 404.256,Z 108.256,A -85,B 0,C 180,E1 -10992.042,E2 -10992.042} C_VEL
LIN {X 0,Y 404.205,Z 108.257,A -85,B 0,C 180,E1 -10995.118,E2 -10995.118} C_VEL
LIN {X 0,Y 404.207,Z 108.258,A -85,B 0,C 180,E1 -10998.238,E2 -10998.238} C_VEL
LIN {X 0,Y 404.159,Z 108.267,A -85,B 0,C 180,E1 -11001.418,E2 -11001.418} C_VEL
LIN {X 0,Y 404.176,Z 108.261,A -85,B 0,C 180,E1 -11004.666,E2 -11004.666} C_VEL
LIN {X 0,Y 404.195,Z 108.259,A -85,B 0,C 180,E1 -11008,E2 -11008} C_VEL
LIN {X 0,Y 404.139,Z 108.268,A -85,B 0,C 180,E1 -11011.558,E2 -11011.558} C_VEL
LIN {X 0,Y 404.183,Z 108.265,A -85,B 0,C 180,E1 -11015.017,E2 -11015.017} C_VEL
LIN {X 0,Y 404.151,Z 108.267,A -85,B 0,C 180,E1 -11018.758,E2 -11018.758} C_VEL
LIN {X 0,Y 404.123,Z 108.268,A -85,B 0,C 180,E1 -11021.6,E2 -11021.6} C_VEL
LIN {X 0,Y 404.146,Z 108.267,A -85,B 0,C 180,E1 -11024.522,E2 -11024.522} C_VEL
LIN {X 0,Y 404.133,Z 108.267,A -85,B 0,C 180,E1 -11027.295,E2 -11027.295} C_VEL
LIN {X 0,Y 404.155,Z 108.264,A -85,B 0,C 180,E1 -11029.954,E2 -11029.954} C_VEL
LIN {X 0,Y 404.136,Z 108.267,A -85,B 0,C 180,E1 -11033.126,E2 -11033.126} C_VEL
LIN {X 0,Y 404.146,Z 108.268,A -85,B 0,C 180,E1 -11036.188,E2 -11036.188} C_VEL
LIN {X 0,Y 404.146,Z 108.265,A -85,B 0,C 180,E1 -11039.715,E2 -11039.715} C_VEL
LIN {X 0,Y 404.136,Z 108.265,A -85,B 0,C 180,E1 -11043.119,E2 -11043.119} C_VEL
LIN {X 0,Y 404.162,Z 108.265,A -85,B 0,C 180,E1 -11046.425,E2 -11046.425} C_VEL
LIN {X 0,Y 404.199,Z 108.331,A -85,B 0,C 180,E1 -11049.118,E2 -11049.118} C_VEL
LIN {X 0,Y 406.689,Z 120.269,A -85,B 0,C 180,E1 -11051.89,E2 -11051.89} C_VEL
LIN {X 0,Y 407.236,Z 123.278,A -85,B 0,C 180,E1 -11052.569,E2 -11052.569} C_VEL
LIN {X 0,Y 409.172,Z 129.806,A -85,B 0,C 180,E1 -11052.806,E2 -11052.806} C_VEL
LIN {X 0,Y 412.988,Z 148.675,A -85,B 0,C 180,E1 -11053.357,E2 -11053.357} C_VEL
LIN {X 0,Y 411.362,Z 260.628,A -85,B 0,C 180,E1 -11055.341,E2 -11055.341} C_VEL
LIN {X 0,Y 410.917,Z 274.934,A -85,B 0,C 180,E1 -11055.799,E2 -11055.799} C_VEL
LIN {X 0,Y 410.189,Z 288.719,A -85,B 0,C 180,E1 -11056.437,E2 -11056.437} C_VEL
LIN {X 0,Y 409.346,Z 301.572,A -85,B 0,C 180,E1 -11057.23,E2 -11057.23} C_VEL
LIN {X 0,Y 408.44,Z 314.038,A -85,B 0,C 180,E1 -11058.21,E2 -11058.21} C_VEL
LIN {X 0,Y 407.516,Z 325.416,A -85,B 0,C 180,E1 -11059.316,E2 -11059.316} C_VEL
LIN {X 0,Y 406.506,Z 336.611,A -85,B 0,C 180,E1 -11060.643,E2 -11060.643} C_VEL
LIN {X 0,Y 405.627,Z 346.262,A -85,B 0,C 180,E1 -11062.033,E2 -11062.033} C_VEL
LIN {X 0,Y 404.858,Z 354.845,A -85,B 0,C 180,E1 -11063.521,E2 -11063.521} C_VEL
LIN {X 0,Y 404.726,Z 356.126,A -85,B 0,C 180,E1 -11063.766,E2 -11063.766} C_VEL
LIN {X 0,Y 403.765,Z 359.546,A -85,B 0,C 180,E1 -11064.434,E2 -11064.434} C_VEL
LIN {X 0,Y 400.549,Z 364.732,A -85,B 0,C 180,E1 -11065.545,E2 -11065.545} C_VEL
LIN {X 0,Y 397.33,Z 369.32,A -85,B 0,C 180,E1 -11066.721,E2 -11066.721} C_VEL
LIN {X 0,Y 396.382,Z 371.805,A -85,B 0,C 180,E1 -11067.485,E2 -11067.485} C_VEL
LIN {X 0,Y 396.031,Z 377.206,A -85,B 0,C 180,E1 -11069.492,E2 -11069.492} C_VEL
LIN {X 0,Y 395.863,Z 380.267,A -85,B 0,C 180,E1 -11071.017,E2 -11071.017} C_VEL
LIN {X 0,Y 395.753,Z 383.133,A -85,B 0,C 180,E1 -11073.054,E2 -11073.054} C_VEL
LIN {X 0,Y 395.774,Z 384.647,A -85,B 0,C 180,E1 -11075.094,E2 -11075.094} C_VEL
LIN {X 0,Y 395.823,Z 384.908,A -85,B 0,C 180,E1 -11076.116,E2 -11076.116} C_VEL
LIN {X 0,Y 395.687,Z 384.443,A -85,B 0,C 180,E1 -11078.169,E2 -11078.169} C_VEL
LIN {X 0,Y 395.757,Z 382.635,A -85,B 0,C 180,E1 -11080.229,E2 -11080.229} C_VEL
LIN {X 0,Y 396.107,Z 379.425,A -85,B 0,C 180,E1 -11082.293,E2 -11082.293} C_VEL
LIN {X 0,Y 396.477,Z 374.679,A -85,B 0,C 180,E1 -11084.369,E2 -11084.369} C_VEL
LIN {X 0,Y 396.926,Z 370.064,A -85,B 0,C 180,E1 -11085.929,E2 -11085.929} C_VEL
LIN {X 0,Y 397.683,Z 363.325,A -85,B 0,C 180,E1 -11087.749,E2 -11087.749} C_VEL
LIN {X 0,Y 398.644,Z 354.888,A -85,B 0,C 180,E1 -11089.571,E2 -11089.571} C_VEL
LIN {X 0,Y 399.706,Z 346.024,A -85,B 0,C 180,E1 -11091.133,E2 -11091.133} C_VEL
LIN {X 0,Y 400.893,Z 335.298,A -85,B 0,C 180,E1 -11092.686,E2 -11092.686} C_VEL
LIN {X 0,Y 402.146,Z 324.392,A -85,B 0,C 180,E1 -11093.974,E2 -11093.974} C_VEL
LIN {X 0,Y 403.437,Z 312.363,A -85,B 0,C 180,E1 -11095.132,E2 -11095.132} C_VEL
LIN {X 0,Y 404.433,Z 300.924,A -85,B 0,C 180,E1 -11096.026,E2 -11096.026} C_VEL
LIN {X 0,Y 405.549,Z 287.452,A -85,B 0,C 180,E1 -11096.85,E2 -11096.85} C_VEL
LIN {X 0,Y 406.334,Z 273.443,A -85,B 0,C 180,E1 -11097.49,E2 -11097.49} C_VEL
LIN {X 0,Y 406.904,Z 259.489,A -85,B 0,C 180,E1 -11097.916,E2 -11097.916} C_VEL
LIN {X 0,Y 408.939,Z 151.877,A -85,B 0,C 180,E1 -11099.856,E2 -11099.856} C_VEL
LIN {X 0,Y 407.461,Z 144.104,A -85,B 0,C 180,E1 -11100.108,E2 -11100.108} C_VEL
LIN {X 0,Y 405.087,Z 134.95,A -85,B 0,C 180,E1 -11100.452,E2 -11100.452} C_VEL
LIN {X 0,Y 400.407,Z 123.658,A -85,B 0,C 180,E1 -11101.024,E2 -11101.024} C_VEL
LIN {X 0,Y 397.854,Z 112.287,A -85,B 0,C 180,E1 -11103.876,E2 -11103.876} C_VEL
LIN {X 0,Y 397.122,Z 109.141,A -85,B 0,C 180,E1 -11104.725,E2 -11104.725} C_VEL
LIN {X 0,Y 397.087,Z 109.148,A -85,B 0,C 180,E1 -11108.277,E2 -11108.277} C_VEL
LIN {X 0,Y 397.051,Z 109.154,A -85,B 0,C 180,E1 -11111.976,E2 -11111.976} C_VEL
LIN {X 0,Y 397.086,Z 109.142,A -85,B 0,C 180,E1 -11115.069,E2 -11115.069} C_VEL
LIN {X 0,Y 397.052,Z 109.151,A -85,B 0,C 180,E1 -11118.023,E2 -11118.023} C_VEL
LIN {X 0,Y 397.091,Z 109.145,A -85,B 0,C 180,E1 -11121.723,E2 -11121.723} C_VEL
LIN {X 0,Y 397.118,Z 109.144,A -85,B 0,C 180,E1 -11125.506,E2 -11125.506} C_VEL
LIN {X 0,Y 397.079,Z 109.148,A -85,B 0,C 180,E1 -11129.117,E2 -11129.117} C_VEL
LIN {X 0,Y 397.093,Z 109.148,A -85,B 0,C 180,E1 -11132.602,E2 -11132.602} C_VEL
LIN {X 0,Y 397.112,Z 109.142,A -85,B 0,C 180,E1 -11135.98,E2 -11135.98} C_VEL
LIN {X 0,Y 397.14,Z 109.138,A -85,B 0,C 180,E1 -11139.704,E2 -11139.704} C_VEL
LIN {X 0,Y 397.183,Z 109.134,A -85,B 0,C 180,E1 -11142.845,E2 -11142.845} C_VEL
LIN {X 0,Y 397.23,Z 109.124,A -85,B 0,C 180,E1 -11146.703,E2 -11146.703} C_VEL
LIN {X 0,Y 397.217,Z 109.13,A -85,B 0,C 180,E1 -11149.809,E2 -11149.809} C_VEL
LIN {X 0,Y 397.319,Z 109.116,A -85,B 0,C 180,E1 -11152.887,E2 -11152.887} C_VEL
LIN {X 0,Y 397.248,Z 109.122,A -85,B 0,C 180,E1 -11154.925,E2 -11154.925} C_VEL
LIN {X 0,Y 397.448,Z 109.102,A -85,B 0,C 180,E1 -11157.973,E2 -11157.973} C_VEL
LIN {X 0,Y 397.577,Z 109.083,A -85,B 0,C 180,E1 -11160,E2 -11160} C_VEL
LIN {X 0,Y 397.368,Z 109.109,A -85,B 0,C 180,E1 -11163.041,E2 -11163.041} C_VEL
LIN {X 0,Y 397.333,Z 109.108,A -85,B 0,C 180,E1 -11166.092,E2 -11166.092} C_VEL
LIN {X 0,Y 397.236,Z 109.128,A -85,B 0,C 180,E1 -11169.162,E2 -11169.162} C_VEL
LIN {X 0,Y 397.22,Z 109.125,A -85,B 0,C 180,E1 -11172.258,E2 -11172.258} C_VEL
LIN {X 0,Y 397.18,Z 109.13,A -85,B 0,C 180,E1 -11175.392,E2 -11175.392} C_VEL
LIN {X 0,Y 397.163,Z 109.135,A -85,B 0,C 180,E1 -11178.573,E2 -11178.573} C_VEL
LIN {X 0,Y 397.098,Z 109.141,A -85,B 0,C 180,E1 -11181.818,E2 -11181.818} C_VEL
LIN {X 0,Y 397.157,Z 109.132,A -85,B 0,C 180,E1 -11185.131,E2 -11185.131} C_VEL
LIN {X 0,Y 397.162,Z 109.133,A -85,B 0,C 180,E1 -11187.776,E2 -11187.776} C_VEL
LIN {X 0,Y 397.08,Z 109.149,A -85,B 0,C 180,E1 -11190.882,E2 -11190.882} C_VEL
LIN {X 0,Y 397.126,Z 109.145,A -85,B 0,C 180,E1 -11194.493,E2 -11194.493} C_VEL
LIN {X 0,Y 397.1,Z 109.142,A -85,B 0,C 180,E1 -11198.275,E2 -11198.275} C_VEL
LIN {X 0,Y 397.089,Z 109.14,A -85,B 0,C 180,E1 -11200.909,E2 -11200.909} C_VEL
LIN {X 0,Y 397.101,Z 109.141,A -85,B 0,C 180,E1 -11203.648,E2 -11203.648} C_VEL
LIN {X 0,Y 397.103,Z 109.147,A -85,B 0,C 180,E1 -11206.521,E2 -11206.521} C_VEL
LIN {X 0,Y 397.115,Z 109.142,A -85,B 0,C 180,E1 -11210.423,E2 -11210.423} C_VEL
LIN {X 0,Y 397.109,Z 109.141,A -85,B 0,C 180,E1 -11214.265,E2 -11214.265} C_VEL
LIN {X 0,Y 397.115,Z 109.134,A -85,B 0,C 180,E1 -11216.727,E2 -11216.727} C_VEL
LIN {X 0,Y 397.107,Z 109.165,A -85,B 0,C 180,E1 -11218.347,E2 -11218.347} C_VEL
LIN {X 0,Y 400.667,Z 123.548,A -85,B 0,C 180,E1 -11221.732,E2 -11221.732} C_VEL
LIN {X 0,Y 402.556,Z 133.173,A -85,B 0,C 180,E1 -11223.865,E2 -11223.865} C_VEL
LIN {X 0,Y 402.034,Z 139.825,A -85,B 0,C 180,E1 -11225.151,E2 -11225.151} C_VEL
LIN {X 0,Y 407.793,Z 167.637,A -85,B 0,C 180,E1 -11226.095,E2 -11226.095} C_VEL
LIN {X 0,Y 408.62,Z 172.455,A -85,B 0,C 180,E1 -11226.244,E2 -11226.244} C_VEL
LIN {X 0,Y 406.633,Z 277.885,A -85,B 0,C 180,E1 -11228.153,E2 -11228.153} C_VEL
LIN {X 0,Y 405.873,Z 292.354,A -85,B 0,C 180,E1 -11228.61,E2 -11228.61} C_VEL
LIN {X 0,Y 404.835,Z 306.786,A -85,B 0,C 180,E1 -11229.285,E2 -11229.285} C_VEL
LIN {X 0,Y 403.73,Z 320.549,A -85,B 0,C 180,E1 -11230.164,E2 -11230.164} C_VEL
LIN {X 0,Y 402.56,Z 332.743,A -85,B 0,C 180,E1 -11231.157,E2 -11231.157} C_VEL
LIN {X 0,Y 401.297,Z 344.014,A -85,B 0,C 180,E1 -11232.284,E2 -11232.284} C_VEL
LIN {X 0,Y 399.989,Z 355.365,A -85,B 0,C 180,E1 -11233.672,E2 -11233.672} C_VEL
LIN {X 0,Y 398.793,Z 365.516,A -85,B 0,C 180,E1 -11235.195,E2 -11235.195} C_VEL
LIN {X 0,Y 397.874,Z 373.95,A -85,B 0,C 180,E1 -11236.725,E2 -11236.725} C_VEL
LIN {X 0,Y 397.204,Z 380.986,A -85,B 0,C 180,E1 -11238.259,E2 -11238.259} C_VEL
LIN {X 0,Y 396.603,Z 386.819,A -85,B 0,C 180,E1 -11239.793,E2 -11239.793} C_VEL
LIN {X 0,Y 396.089,Z 393.074,A -85,B 0,C 180,E1 -11241.839,E2 -11241.839} C_VEL
LIN {X 0,Y 395.86,Z 397.688,A -85,B 0,C 180,E1 -11243.885,E2 -11243.885} C_VEL
LIN {X 0,Y 395.748,Z 400.832,A -85,B 0,C 180,E1 -11245.926,E2 -11245.926} C_VEL
LIN {X 0,Y 395.75,Z 402.613,A -85,B 0,C 180,E1 -11247.964,E2 -11247.964} C_VEL
LIN {X 0,Y 395.759,Z 403.06,A -85,B 0,C 180,E1 -11250,E2 -11250} C_VEL
LIN {X 0,Y 395.758,Z 402.176,A -85,B 0,C 180,E1 -11252.035,E2 -11252.035} C_VEL
LIN {X 0,Y 395.747,Z 399.937,A -85,B 0,C 180,E1 -11254.073,E2 -11254.073} C_VEL
LIN {X 0,Y 395.82,Z 396.283,A -85,B 0,C 180,E1 -11256.115,E2 -11256.115} C_VEL
LIN {X 0,Y 396.054,Z 391.104,A -85,B 0,C 180,E1 -11258.161,E2 -11258.161} C_VEL
LIN {X 0,Y 396.325,Z 386.073,A -85,B 0,C 180,E1 -11259.698,E2 -11259.698} C_VEL
LIN {X 0,Y 396.888,Z 378.867,A -85,B 0,C 180,E1 -11261.491,E2 -11261.491} C_VEL
LIN {X 0,Y 397.537,Z 371.312,A -85,B 0,C 180,E1 -11263.027,E2 -11263.027} C_VEL
LIN {X 0,Y 398.231,Z 362.222,A -85,B 0,C 180,E1 -11264.565,E2 -11264.565} C_VEL
LIN {X 0,Y 399.278,Z 351.213,A -85,B 0,C 180,E1 -11266.095,E2 -11266.095} C_VEL
LIN {X 0,Y 400.368,Z 340.023,A -85,B 0,C 180,E1 -11267.362,E2 -11267.362} C_VEL
LIN {X 0,Y 401.449,Z 327.774,A -85,B 0,C 180,E1 -11268.49,E2 -11268.49} C_VEL
LIN {X 0,Y 402.436,Z 314.931,A -85,B 0,C 180,E1 -11269.432,E2 -11269.432} C_VEL
LIN {X 0,Y 403.278,Z 301.814,A -85,B 0,C 180,E1 -11270.178,E2 -11270.178} C_VEL
LIN {X 0,Y 404.037,Z 287.873,A -85,B 0,C 180,E1 -11270.757,E2 -11270.757} C_VEL
LIN {X 0,Y 404.573,Z 272.814,A -85,B 0,C 180,E1 -11271.161,E2 -11271.161} C_VEL
LIN {X 0,Y 406.133,Z 171.677,A -85,B 0,C 180,E1 -11272.956,E2 -11272.956} C_VEL
LIN {X 0,Y 400.677,Z 139.818,A -85,B 0,C 180,E1 -11273.854,E2 -11273.854} C_VEL
LIN {X 0,Y 401.448,Z 130.304,A -85,B 0,C 180,E1 -11275.676,E2 -11275.676} C_VEL
LIN {X 0,Y 400.269,Z 123.155,A -85,B 0,C 180,E1 -11277.162,E2 -11277.162} C_VEL
LIN {X 0,Y 397.135,Z 109.144,A -85,B 0,C 180,E1 -11280.264,E2 -11280.264} C_VEL
LIN {X 0,Y 397.118,Z 109.142,A -85,B 0,C 180,E1 -11283.718,E2 -11283.718} C_VEL
LIN {X 0,Y 397.093,Z 109.143,A -85,B 0,C 180,E1 -11287.209,E2 -11287.209} C_VEL
LIN {X 0,Y 397.1,Z 109.144,A -85,B 0,C 180,E1 -11290.445,E2 -11290.445} C_VEL
LIN {X 0,Y 397.103,Z 109.146,A -85,B 0,C 180,E1 -11293.648,E2 -11293.648} C_VEL
LIN {X 0,Y 397.161,Z 109.135,A -85,B 0,C 180,E1 -11296.512,E2 -11296.512} C_VEL
LIN {X 0,Y 397.112,Z 109.146,A -85,B 0,C 180,E1 -11299.552,E2 -11299.552} C_VEL
LIN {X 0,Y 397.097,Z 109.144,A -85,B 0,C 180,E1 -11303.005,E2 -11303.005} C_VEL
LIN {X 0,Y 397.117,Z 109.14,A -85,B 0,C 180,E1 -11306.282,E2 -11306.282} C_VEL
LIN {X 0,Y 397.104,Z 109.141,A -85,B 0,C 180,E1 -11310.135,E2 -11310.135} C_VEL
LIN {X 0,Y 397.193,Z 109.131,A -85,B 0,C 180,E1 -11312.61,E2 -11312.61} C_VEL
LIN {X 0,Y 397.132,Z 109.138,A -85,B 0,C 180,E1 -11315.982,E2 -11315.982} C_VEL
LIN {X 0,Y 397.137,Z 109.138,A -85,B 0,C 180,E1 -11319.705,E2 -11319.705} C_VEL
LIN {X 0,Y 397.181,Z 109.138,A -85,B 0,C 180,E1 -11322.845,E2 -11322.845} C_VEL
LIN {X 0,Y 397.227,Z 109.132,A -85,B 0,C 180,E1 -11326.703,E2 -11326.703} C_VEL
LIN {X 0,Y 397.217,Z 109.127,A -85,B 0,C 180,E1 -11329.809,E2 -11329.809} C_VEL
LIN {X 0,Y 397.349,Z 109.114,A -85,B 0,C 180,E1 -11332.888,E2 -11332.888} C_VEL
LIN {X 0,Y 397.252,Z 109.125,A -85,B 0,C 180,E1 -11334.925,E2 -11334.925} C_VEL
LIN {X 0,Y 397.448,Z 109.101,A -85,B 0,C 180,E1 -11337.973,E2 -11337.973} C_VEL
LIN {X 0,Y 397.578,Z 109.086,A -85,B 0,C 180,E1 -11340,E2 -11340} C_VEL
LIN {X 0,Y 397.374,Z 109.108,A -85,B 0,C 180,E1 -11343.042,E2 -11343.042} C_VEL
LIN {X 0,Y 397.323,Z 109.116,A -85,B 0,C 180,E1 -11346.517,E2 -11346.517} C_VEL
LIN {X 0,Y 397.251,Z 109.123,A -85,B 0,C 180,E1 -11349.162,E2 -11349.162} C_VEL
LIN {X 0,Y 397.219,Z 109.13,A -85,B 0,C 180,E1 -11352.258,E2 -11352.258} C_VEL
LIN {X 0,Y 397.178,Z 109.135,A -85,B 0,C 180,E1 -11355.392,E2 -11355.392} C_VEL
LIN {X 0,Y 397.16,Z 109.134,A -85,B 0,C 180,E1 -11358.574,E2 -11358.574} C_VEL
LIN {X 0,Y 397.108,Z 109.145,A -85,B 0,C 180,E1 -11361.818,E2 -11361.818} C_VEL
LIN {X 0,Y 397.152,Z 109.142,A -85,B 0,C 180,E1 -11365.513,E2 -11365.513} C_VEL
LIN {X 0,Y 397.121,Z 109.139,A -85,B 0,C 180,E1 -11368.544,E2 -11368.544} C_VEL
LIN {X 0,Y 397.078,Z 109.145,A -85,B 0,C 180,E1 -11372.072,E2 -11372.072} C_VEL
LIN {X 0,Y 397.118,Z 109.142,A -85,B 0,C 180,E1 -11375.504,E2 -11375.504} C_VEL
LIN {X 0,Y 397.127,Z 109.143,A -85,B 0,C 180,E1 -11378.861,E2 -11378.861} C_VEL
LIN {X 0,Y 397.068,Z 109.147,A -85,B 0,C 180,E1 -11382.268,E2 -11382.268} C_VEL
LIN {X 0,Y 397.087,Z 109.147,A -85,B 0,C 180,E1 -11385.069,E2 -11385.069} C_VEL
LIN {X 0,Y 397.063,Z 109.147,A -85,B 0,C 180,E1 -11388.022,E2 -11388.022} C_VEL
LIN {X 0,Y 397.125,Z 109.14,A -85,B 0,C 180,E1 -11391.14,E2 -11391.14} C_VEL
LIN {X 0,Y 397.12,Z 109.146,A -85,B 0,C 180,E1 -11394.497,E2 -11394.497} C_VEL
LIN {X 0,Y 397.08,Z 109.146,A -85,B 0,C 180,E1 -11397.929,E2 -11397.929} C_VEL
LIN {X 0,Y 397.12,Z 109.146,A -85,B 0,C 180,E1 -11400.296,E2 -11400.296} C_VEL
LIN {X 0,Y 397.096,Z 109.144,A -85,B 0,C 180,E1 -11403.739,E2 -11403.739} C_VEL
LIN {X 0,Y 397.106,Z 109.141,A -85,B 0,C 180,E1 -11407.086,E2 -11407.086} C_VEL
LIN {X 0,Y 397.133,Z 109.145,A -85,B 0,C 180,E1 -11408.797,E2 -11408.797} C_VEL
LIN {X 0,Y 399.713,Z 121.448,A -85,B 0,C 180,E1 -11411.708,E2 -11411.708} C_VEL
LIN {X 0,Y 400.113,Z 123.491,A -85,B 0,C 180,E1 -11412.18,E2 -11412.18} C_VEL
LIN {X 0,Y 402.756,Z 131.798,A -85,B 0,C 180,E1 -11412.488,E2 -11412.488} C_VEL
LIN {X 0,Y 406.406,Z 150.12,A -85,B 0,C 180,E1 -11413.032,E2 -11413.032} C_VEL
LIN {X 0,Y 404.707,Z 259.876,A -85,B 0,C 180,E1 -11414.998,E2 -11414.998} C_VEL
LIN {X 0,Y 404.241,Z 273.766,A -85,B 0,C 180,E1 -11415.431,E2 -11415.431} C_VEL
LIN {X 0,Y 403.481,Z 287.897,A -85,B 0,C 180,E1 -11416.079,E2 -11416.079} C_VEL
LIN {X 0,Y 402.628,Z 300.962,A -85,B 0,C 180,E1 -11416.884,E2 -11416.884} C_VEL
LIN {X 0,Y 401.663,Z 313.581,A -85,B 0,C 180,E1 -11417.88,E2 -11417.88} C_VEL
LIN {X 0,Y 400.673,Z 325.184,A -85,B 0,C 180,E1 -11419.016,E2 -11419.016} C_VEL
LIN {X 0,Y 399.636,Z 336.296,A -85,B 0,C 180,E1 -11420.346,E2 -11420.346} C_VEL
LIN {X 0,Y 398.624,Z 346.88,A -85,B 0,C 180,E1 -11421.892,E2 -11421.892} C_VEL
LIN {X 0,Y 397.846,Z 355.387,A -85,B 0,C 180,E1 -11423.407,E2 -11423.407} C_VEL
LIN {X 0,Y 397.071,Z 363.557,A -85,B 0,C 180,E1 -11425.177,E2 -11425.177} C_VEL
LIN {X 0,Y 396.41,Z 370.135,A -85,B 0,C 180,E1 -11426.951,E2 -11426.951} C_VEL
LIN {X 0,Y 396.382,Z 371.805,A -85,B 0,C 180,E1 -11427.485,E2 -11427.485} C_VEL
LIN {X 0,Y 395.456,Z 374.139,A -85,B 0,C 180,E1 -11428.264,E2 -11428.264} C_VEL
LIN {X 0,Y 392.368,Z 377.518,A -85,B 0,C 180,E1 -11429.546,E2 -11429.546} C_VEL
LIN {X 0,Y 389.889,Z 379.77,A -85,B 0,C 180,E1 -11430.602,E2 -11430.602} C_VEL
LIN {X 0,Y 388.761,Z 381.441,A -85,B 0,C 180,E1 -11431.574,E2 -11431.574} C_VEL
LIN {X 0,Y 388.734,Z 381.591,A -85,B 0,C 180,E1 -11431.715,E2 -11431.715} C_VEL
LIN {X 0,Y 388.657,Z 383.375,A -85,B 0,C 180,E1 -11433.11,E2 -11433.11} C_VEL
LIN {X 0,Y 388.678,Z 384.844,A -85,B 0,C 180,E1 -11435.187,E2 -11435.187} C_VEL
LIN {X 0,Y 388.723,Z 385.083,A -85,B 0,C 180,E1 -11436.228,E2 -11436.228} C_VEL
LIN {X 0,Y 388.604,Z 384.573,A -85,B 0,C 180,E1 -11438.319,E2 -11438.319} C_VEL
LIN {X 0,Y 388.703,Z 382.717,A -85,B 0,C 180,E1 -11440.417,E2 -11440.417} C_VEL
LIN {X 0,Y 389.07,Z 379.441,A -85,B 0,C 180,E1 -11442.519,E2 -11442.519} C_VEL
LIN {X 0,Y 389.464,Z 374.641,A -85,B 0,C 180,E1 -11444.634,E2 -11444.634} C_VEL
LIN {X 0,Y 389.977,Z 369.988,A -85,B 0,C 180,E1 -11446.221,E2 -11446.221} C_VEL
LIN {X 0,Y 390.757,Z 363.175,A -85,B 0,C 180,E1 -11448.075,E2 -11448.075} C_VEL
LIN {X 0,Y 391.642,Z 356.033,A -85,B 0,C 180,E1 -11449.662,E2 -11449.662} C_VEL
LIN {X 0,Y 392.684,Z 347.79,A -85,B 0,C 180,E1 -11451.181,E2 -11451.181} C_VEL
LIN {X 0,Y 393.81,Z 338.806,A -85,B 0,C 180,E1 -11452.563,E2 -11452.563} C_VEL
LIN {X 0,Y 394.988,Z 328.586,A -85,B 0,C 180,E1 -11453.878,E2 -11453.878} C_VEL
LIN {X 0,Y 396.265,Z 317.496,A -85,B 0,C 180,E1 -11455.052,E2 -11455.052} C_VEL
LIN {X 0,Y 397.435,Z 305.597,A -85,B 0,C 180,E1 -11456.082,E2 -11456.082} C_VEL
LIN {X 0,Y 398.722,Z 292.098,A -85,B 0,C 180,E1 -11456.993,E2 -11456.993} C_VEL
LIN {X 0,Y 399.534,Z 278.893,A -85,B 0,C 180,E1 -11457.678,E2 -11457.678} C_VEL
LIN {X 0,Y 400.225,Z 264.644,A -85,B 0,C 180,E1 -11458.195,E2 -11458.195} C_VEL
LIN {X 0,Y 400.693,Z 246.874,A -85,B 0,C 180,E1 -11458.581,E2 -11458.581} C_VEL
LIN {X 0,Y 402.558,Z 152.224,A -85,B 0,C 180,E1 -11460.296,E2 -11460.296} C_VEL
LIN {X 0,Y 399.196,Z 137.903,A -85,B 0,C 180,E1 -11460.821,E2 -11460.821} C_VEL
LIN {X 0,Y 393.253,Z 123.832,A -85,B 0,C 180,E1 -11461.563,E2 -11461.563} C_VEL
LIN {X 0,Y 390.563,Z 112.063,A -85,B 0,C 180,E1 -11464.595,E2 -11464.595} C_VEL
LIN {X 0,Y 390.083,Z 110.018,A -85,B 0,C 180,E1 -11465.172,E2 -11465.172} C_VEL
LIN {X 0,Y 390.055,Z 110.023,A -85,B 0,C 180,E1 -11469.097,E2 -11469.097} C_VEL
LIN {X 0,Y 390.03,Z 110.026,A -85,B 0,C 180,E1 -11472.372,E2 -11472.372} C_VEL
LIN {X 0,Y 390.041,Z 110.017,A -85,B 0,C 180,E1 -11475.353,E2 -11475.353} C_VEL
LIN {X 0,Y 390.016,Z 110.027,A -85,B 0,C 180,E1 -11478.184,E2 -11478.184} C_VEL
LIN {X 0,Y 390.058,Z 110.01,A -85,B 0,C 180,E1 -11480.903,E2 -11480.903} C_VEL
LIN {X 0,Y 390.07,Z 110.018,A -85,B 0,C 180,E1 -11484.791,E2 -11484.791} C_VEL
LIN {X 0,Y 390.024,Z 110.026,A -85,B 0,C 180,E1 -11488.495,E2 -11488.495} C_VEL
LIN {X 0,Y 390.03,Z 110.024,A -85,B 0,C 180,E1 -11492.063,E2 -11492.063} C_VEL
LIN {X 0,Y 390.043,Z 110.023,A -85,B 0,C 180,E1 -11495.517,E2 -11495.517} C_VEL
LIN {X 0,Y 390.056,Z 110.023,A -85,B 0,C 180,E1 -11498.878,E2 -11498.878} C_VEL
LIN {X 0,Y 390.112,Z 110.008,A -85,B 0,C 180,E1 -11502.166,E2 -11502.166} C_VEL
LIN {X 0,Y 390.144,Z 110.007,A -85,B 0,C 180,E1 -11505.392,E2 -11505.392} C_VEL
LIN {X 0,Y 390.149,Z 110.013,A -85,B 0,C 180,E1 -11508.571,E2 -11508.571} C_VEL
LIN {X 0,Y 390.259,Z 109.991,A -85,B 0,C 180,E1 -11512.084,E2 -11512.084} C_VEL
LIN {X 0,Y 390.219,Z 109.998,A -85,B 0,C 180,E1 -11514.833,E2 -11514.833} C_VEL
LIN {X 0,Y 390.417,Z 109.977,A -85,B 0,C 180,E1 -11517.937,E2 -11517.937} C_VEL
LIN {X 0,Y 390.547,Z 109.958,A -85,B 0,C 180,E1 -11520,E2 -11520} C_VEL
LIN {X 0,Y 390.303,Z 109.989,A -85,B 0,C 180,E1 -11523.096,E2 -11523.096} C_VEL
LIN {X 0,Y 390.287,Z 109.985,A -85,B 0,C 180,E1 -11526.202,E2 -11526.202} C_VEL
LIN {X 0,Y 390.194,Z 110.007,A -85,B 0,C 180,E1 -11529.329,E2 -11529.329} C_VEL
LIN {X 0,Y 390.171,Z 110.003,A -85,B 0,C 180,E1 -11532.483,E2 -11532.483} C_VEL
LIN {X 0,Y 390.14,Z 110.003,A -85,B 0,C 180,E1 -11535.677,E2 -11535.677} C_VEL
LIN {X 0,Y 390.106,Z 110.016,A -85,B 0,C 180,E1 -11538.922,E2 -11538.922} C_VEL
LIN {X 0,Y 390.041,Z 110.02,A -85,B 0,C 180,E1 -11542.234,E2 -11542.234} C_VEL
LIN {X 0,Y 390.12,Z 110.01,A -85,B 0,C 180,E1 -11545.743,E2 -11545.743} C_VEL
LIN {X 0,Y 390.059,Z 110.018,A -85,B 0,C 180,E1 -11549.109,E2 -11549.109} C_VEL
LIN {X 0,Y 390.043,Z 110.021,A -85,B 0,C 180,E1 -11552.721,E2 -11552.721} C_VEL
LIN {X 0,Y 390.056,Z 110.017,A -85,B 0,C 180,E1 -11555.825,E2 -11555.825} C_VEL
LIN {X 0,Y 390.067,Z 110.007,A -85,B 0,C 180,E1 -11559.218,E2 -11559.218} C_VEL
LIN {X 0,Y 390.043,Z 110.027,A -85,B 0,C 180,E1 -11562.374,E2 -11562.374} C_VEL
LIN {X 0,Y 390.045,Z 110.018,A -85,B 0,C 180,E1 -11565.354,E2 -11565.354} C_VEL
LIN {X 0,Y 390.032,Z 110.028,A -85,B 0,C 180,E1 -11568.187,E2 -11568.187} C_VEL
LIN {X 0,Y 390.092,Z 110.014,A -85,B 0,C 180,E1 -11570.908,E2 -11570.908} C_VEL
LIN {X 0,Y 390.086,Z 110.014,A -85,B 0,C 180,E1 -11574.793,E2 -11574.793} C_VEL
LIN {X 0,Y 390.034,Z 110.027,A -85,B 0,C 180,E1 -11577.875,E2 -11577.875} C_VEL
LIN {X 0,Y 393.124,Z 122.276,A -85,B 0,C 180,E1 -11580.847,E2 -11580.847} C_VEL
LIN {X 0,Y 395.475,Z 133.125,A -85,B 0,C 180,E1 -11583.338,E2 -11583.338} C_VEL
LIN {X 0,Y 395.711,Z 135.851,A -85,B 0,C 180,E1 -11583.924,E2 -11583.924} C_VEL
LIN {X 0,Y 395.321,Z 139.482,A -85,B 0,C 180,E1 -11584.648,E2 -11584.648} C_VEL
LIN {X 0,Y 401.429,Z 168.634,A -85,B 0,C 180,E1 -11585.673,E2 -11585.673} C_VEL
LIN {X 0,Y 402.197,Z 174.445,A -85,B 0,C 180,E1 -11585.84,E2 -11585.84} C_VEL
LIN {X 0,Y 400.201,Z 276.754,A -85,B 0,C 180,E1 -11587.715,E2 -11587.715} C_VEL
LIN {X 0,Y 399.483,Z 290.832,A -85,B 0,C 180,E1 -11588.149,E2 -11588.149} C_VEL
LIN {X 0,Y 398.438,Z 305.053,A -85,B 0,C 180,E1 -11588.802,E2 -11588.802} C_VEL
LIN {X 0,Y 397.267,Z 318.679,A -85,B 0,C 180,E1 -11589.655,E2 -11589.655} C_VEL
LIN {X 0,Y 395.964,Z 331.587,A -85,B 0,C 180,E1 -11590.696,E2 -11590.696} C_VEL
LIN {X 0,Y 394.68,Z 343.03,A -85,B 0,C 180,E1 -11591.843,E2 -11591.843} C_VEL
LIN {X 0,Y 393.395,Z 353.55,A -85,B 0,C 180,E1 -11593.124,E2 -11593.124} C_VEL
LIN {X 0,Y 392.088,Z 364.013,A -85,B 0,C 180,E1 -11594.669,E2 -11594.669} C_VEL
LIN {X 0,Y 391.136,Z 372.373,A -85,B 0,C 180,E1 -11596.17,E2 -11596.17} C_VEL
LIN {X 0,Y 390.325,Z 379.868,A -85,B 0,C 180,E1 -11597.786,E2 -11597.786} C_VEL
LIN {X 0,Y 389.557,Z 386.787,A -85,B 0,C 180,E1 -11599.606,E2 -11599.606} C_VEL
LIN {X 0,Y 389.039,Z 393.01,A -85,B 0,C 180,E1 -11601.69,E2 -11601.69} C_VEL
LIN {X 0,Y 388.776,Z 397.588,A -85,B 0,C 180,E1 -11603.773,E2 -11603.773} C_VEL
LIN {X 0,Y 388.672,Z 400.709,A -85,B 0,C 180,E1 -11605.852,E2 -11605.852} C_VEL
LIN {X 0,Y 388.646,Z 402.466,A -85,B 0,C 180,E1 -11607.927,E2 -11607.927} C_VEL
LIN {X 0,Y 388.689,Z 402.892,A -85,B 0,C 180,E1 -11610,E2 -11610} C_VEL
LIN {X 0,Y 388.655,Z 401.984,A -85,B 0,C 180,E1 -11612.072,E2 -11612.072} C_VEL
LIN {X 0,Y 388.67,Z 399.723,A -85,B 0,C 180,E1 -11614.148,E2 -11614.148} C_VEL
LIN {X 0,Y 388.75,Z 396.044,A -85,B 0,C 180,E1 -11616.227,E2 -11616.227} C_VEL
LIN {X 0,Y 388.978,Z 390.837,A -85,B 0,C 180,E1 -11618.311,E2 -11618.311} C_VEL
LIN {X 0,Y 389.278,Z 385.778,A -85,B 0,C 180,E1 -11619.876,E2 -11619.876} C_VEL
LIN {X 0,Y 389.882,Z 378.54,A -85,B 0,C 180,E1 -11621.7,E2 -11621.7} C_VEL
LIN {X 0,Y 390.542,Z 370.948,A -85,B 0,C 180,E1 -11623.264,E2 -11623.264} C_VEL
LIN {X 0,Y 391.292,Z 361.818,A -85,B 0,C 180,E1 -11624.829,E2 -11624.829} C_VEL
LIN {X 0,Y 392.206,Z 352.729,A -85,B 0,C 180,E1 -11626.126,E2 -11626.126} C_VEL
LIN {X 0,Y 393.293,Z 341.879,A -85,B 0,C 180,E1 -11627.416,E2 -11627.416} C_VEL
LIN {X 0,Y 394.415,Z 330.007,A -85,B 0,C 180,E1 -11628.573,E2 -11628.573} C_VEL
LIN {X 0,Y 395.504,Z 316.813,A -85,B 0,C 180,E1 -11629.602,E2 -11629.602} C_VEL
LIN {X 0,Y 396.451,Z 303.095,A -85,B 0,C 180,E1 -11630.426,E2 -11630.426} C_VEL
LIN {X 0,Y 397.284,Z 289.38,A -85,B 0,C 180,E1 -11631.025,E2 -11631.025} C_VEL
LIN {X 0,Y 397.802,Z 275.384,A -85,B 0,C 180,E1 -11631.437,E2 -11631.437} C_VEL
LIN {X 0,Y 399.499,Z 172.969,A -85,B 0,C 180,E1 -11633.291,E2 -11633.291} C_VEL
LIN {X 0,Y 393.847,Z 139.582,A -85,B 0,C 180,E1 -11634.266,E2 -11634.266} C_VEL
LIN {X 0,Y 394.545,Z 131.326,A -85,B 0,C 180,E1 -11635.875,E2 -11635.875} C_VEL
LIN {X 0,Y 392.504,Z 120.811,A -85,B 0,C 180,E1 -11638.134,E2 -11638.134} C_VEL
LIN {X 0,Y 390.085,Z 110.021,A -85,B 0,C 180,E1 -11640.595,E2 -11640.595} C_VEL
LIN {X 0,Y 390.068,Z 110.023,A -85,B 0,C 180,E1 -11644.024,E2 -11644.024} C_VEL
LIN {X 0,Y 390.042,Z 110.023,A -85,B 0,C 180,E1 -11647.551,E2 -11647.551} C_VEL
LIN {X 0,Y 390.055,Z 110.019,A -85,B 0,C 180,E1 -11650.821,E2 -11650.821} C_VEL
LIN {X 0,Y 390.059,Z 110.025,A -85,B 0,C 180,E1 -11653.887,E2 -11653.887} C_VEL
LIN {X 0,Y 390.114,Z 110.012,A -85,B 0,C 180,E1 -11656.798,E2 -11656.798} C_VEL
LIN {X 0,Y 390.067,Z 110.024,A -85,B 0,C 180,E1 -11659.562,E2 -11659.562} C_VEL
LIN {X 0,Y 390.041,Z 110.021,A -85,B 0,C 180,E1 -11662.449,E2 -11662.449} C_VEL
LIN {X 0,Y 390.067,Z 110.019,A -85,B 0,C 180,E1 -11665.975,E2 -11665.975} C_VEL
LIN {X 0,Y 390.045,Z 110.022,A -85,B 0,C 180,E1 -11669.869,E2 -11669.869} C_VEL
LIN {X 0,Y 390.112,Z 110.019,A -85,B 0,C 180,E1 -11673.232,E2 -11673.232} C_VEL
LIN {X 0,Y 390.105,Z 110.016,A -85,B 0,C 180,E1 -11676.75,E2 -11676.75} C_VEL
LIN {X 0,Y 390.102,Z 110.013,A -85,B 0,C 180,E1 -11679.983,E2 -11679.983} C_VEL
LIN {X 0,Y 390.137,Z 110.012,A -85,B 0,C 180,E1 -11683.248,E2 -11683.248} C_VEL
LIN {X 0,Y 390.193,Z 110.007,A -85,B 0,C 180,E1 -11686.562,E2 -11686.562} C_VEL
LIN {X 0,Y 390.204,Z 110.007,A -85,B 0,C 180,E1 -11690.671,E2 -11690.671} C_VEL
LIN {X 0,Y 390.323,Z 109.987,A -85,B 0,C 180,E1 -11693.798,E2 -11693.798} C_VEL
LIN {X 0,Y 390.417,Z 109.977,A -85,B 0,C 180,E1 -11697.937,E2 -11697.937} C_VEL
LIN {X 0,Y 390.547,Z 109.961,A -85,B 0,C 180,E1 -11700,E2 -11700} C_VEL
LIN {X 0,Y 390.309,Z 109.988,A -85,B 0,C 180,E1 -11703.097,E2 -11703.097} C_VEL
LIN {X 0,Y 390.282,Z 109.994,A -85,B 0,C 180,E1 -11706.507,E2 -11706.507} C_VEL
LIN {X 0,Y 390.203,Z 110.002,A -85,B 0,C 180,E1 -11709.329,E2 -11709.329} C_VEL
LIN {X 0,Y 390.17,Z 110.006,A -85,B 0,C 180,E1 -11712.483,E2 -11712.483} C_VEL
LIN {X 0,Y 390.138,Z 110.014,A -85,B 0,C 180,E1 -11715.677,E2 -11715.677} C_VEL
LIN {X 0,Y 390.104,Z 110.014,A -85,B 0,C 180,E1 -11718.922,E2 -11718.922} C_VEL
LIN {X 0,Y 390.046,Z 110.021,A -85,B 0,C 180,E1 -11722.234,E2 -11722.234} C_VEL
LIN {X 0,Y 390.119,Z 110.015,A -85,B 0,C 180,E1 -11725.744,E2 -11725.744} C_VEL
LIN {X 0,Y 390.058,Z 110.023,A -85,B 0,C 180,E1 -11729.11,E2 -11729.11} C_VEL
LIN {X 0,Y 390.043,Z 110.023,A -85,B 0,C 180,E1 -11732.722,E2 -11732.722} C_VEL
LIN {X 0,Y 390.055,Z 110.02,A -85,B 0,C 180,E1 -11735.826,E2 -11735.826} C_VEL
LIN {X 0,Y 390.068,Z 110.022,A -85,B 0,C 180,E1 -11739.218,E2 -11739.218} C_VEL
LIN {X 0,Y 390.042,Z 110.023,A -85,B 0,C 180,E1 -11742.374,E2 -11742.374} C_VEL
LIN {X 0,Y 390.044,Z 110.022,A -85,B 0,C 180,E1 -11745.355,E2 -11745.355} C_VEL
LIN {X 0,Y 390.028,Z 110.024,A -85,B 0,C 180,E1 -11748.187,E2 -11748.187} C_VEL
LIN {X 0,Y 390.083,Z 110.019,A -85,B 0,C 180,E1 -11750.907,E2 -11750.907} C_VEL
LIN {X 0,Y 390.086,Z 110.019,A -85,B 0,C 180,E1 -11754.794,E2 -11754.794} C_VEL
LIN {X 0,Y 390.025,Z 110.028,A -85,B 0,C 180,E1 -11758.496,E2 -11758.496} C_VEL
LIN {X 0,Y 390.04,Z 110.026,A -85,B 0,C 180,E1 -11762.064,E2 -11762.064} C_VEL
LIN {X 0,Y 390.056,Z 110.02,A -85,B 0,C 180,E1 -11765.518,E2 -11765.518} C_VEL
LIN {X 0,Y 390.07,Z 110.099,A -85,B 0,C 180,E1 -11768.498,E2 -11768.498} C_VEL
LIN {X 0,Y 392.527,Z 121.246,A -85,B 0,C 180,E1 -11771.199,E2 -11771.199} C_VEL
LIN {X 0,Y 392.949,Z 123.649,A -85,B 0,C 180,E1 -11771.763,E2 -11771.763} C_VEL
LIN {X 0,Y 396.277,Z 133.434,A -85,B 0,C 180,E1 -11772.149,E2 -11772.149} C_VEL
LIN {X 0,Y 399.731,Z 150.84,A -85,B 0,C 180,E1 -11772.677,E2 -11772.677} C_VEL
LIN {X 0,Y 397.989,Z 260.304,A -85,B 0,C 180,E1 -11774.673,E2 -11774.673} C_VEL
LIN {X 0,Y 397.492,Z 274.838,A -85,B 0,C 180,E1 -11775.145,E2 -11775.145} C_VEL
LIN {X 0,Y 396.676,Z 289.293,A -85,B 0,C 180,E1 -11775.835,E2 -11775.835} C_VEL
LIN {X 0,Y 395.767,Z 302.094,A -85,B 0,C 180,E1 -11776.653,E2 -11776.653} C_VEL
LIN {X 0,Y 394.778,Z 314.526,A -85,B 0,C 180,E1 -11777.665,E2 -11777.665} C_VEL
LIN {X 0,Y 393.773,Z 325.99,A -85,B 0,C 180,E1 -11778.821,E2 -11778.821} C_VEL
LIN {X 0,Y 392.652,Z 337.225,A -85,B 0,C 180,E1 -11780.203,E2 -11780.203} C_VEL
LIN {X 0,Y 391.623,Z 347.486,A -85,B 0,C 180,E1 -11781.746,E2 -11781.746} C_VEL
LIN {X 0,Y 390.838,Z 355.92,A -85,B 0,C 180,E1 -11783.288,E2 -11783.288} C_VEL
LIN {X 0,Y 390.022,Z 364.001,A -85,B 0,C 180,E1 -11785.09,E2 -11785.09} C_VEL
LIN {X 0,Y 389.346,Z 370.522,A -85,B 0,C 180,E1 -11786.896,E2 -11786.896} C_VEL
LIN {X 0,Y 388.947,Z 376.312,A -85,B 0,C 180,E1 -11788.965,E2 -11788.965} C_VEL
LIN {X 0,Y 388.789,Z 380.554,A -85,B 0,C 180,E1 -11791.036,E2 -11791.036} C_VEL
LIN {X 0,Y 388.734,Z 381.591,A -85,B 0,C 180,E1 -11791.715,E2 -11791.715} C_VEL
LIN {X 0,Y 388.064,Z 382.799,A -85,B 0,C 180,E1 -11792.561,E2 -11792.561} C_VEL
LIN {X 0,Y 385.251,Z 384.202,A -85,B 0,C 180,E1 -11793.951,E2 -11793.951} C_VEL
LIN {X 0,Y 382.839,Z 384.922,A -85,B 0,C 180,E1 -11795.082,E2 -11795.082} C_VEL
LIN {X 0,Y 381.748,Z 385.201,A -85,B 0,C 180,E1 -11795.958,E2 -11795.958} C_VEL
LIN {X 0,Y 381.628,Z 385.244,A -85,B 0,C 180,E1 -11796.255,E2 -11796.255} C_VEL
LIN {X 0,Y 381.506,Z 384.703,A -85,B 0,C 180,E1 -11798.475,E2 -11798.475} C_VEL
LIN {X 0,Y 381.654,Z 382.79,A -85,B 0,C 180,E1 -11800.611,E2 -11800.611} C_VEL
LIN {X 0,Y 382.05,Z 379.271,A -85,B 0,C 180,E1 -11802.847,E2 -11802.847} C_VEL
LIN {X 0,Y 382.454,Z 374.606,A -85,B 0,C 180,E1 -11804.908,E2 -11804.908} C_VEL
LIN {X 0,Y 382.998,Z 369.9,A -85,B 0,C 180,E1 -11806.525,E2 -11806.525} C_VEL
LIN {X 0,Y 383.862,Z 363.026,A -85,B 0,C 180,E1 -11808.411,E2 -11808.411} C_VEL
LIN {X 0,Y 384.954,Z 354.454,A -85,B 0,C 180,E1 -11810.297,E2 -11810.297} C_VEL
LIN {X 0,Y 386.318,Z 344.633,A -85,B 0,C 180,E1 -11812.04,E2 -11812.04} C_VEL
LIN {X 0,Y 387.519,Z 334.531,A -85,B 0,C 180,E1 -11813.515,E2 -11813.515} C_VEL
LIN {X 0,Y 388.943,Z 323.477,A -85,B 0,C 180,E1 -11814.834,E2 -11814.834} C_VEL
LIN {X 0,Y 390.353,Z 311.143,A -85,B 0,C 180,E1 -11816.03,E2 -11816.03} C_VEL
LIN {X 0,Y 391.515,Z 299.28,A -85,B 0,C 180,E1 -11816.953,E2 -11816.953} C_VEL
LIN {X 0,Y 392.588,Z 286.374,A -85,B 0,C 180,E1 -11817.739,E2 -11817.739} C_VEL
LIN {X 0,Y 393.433,Z 272.539,A -85,B 0,C 180,E1 -11818.363,E2 -11818.363} C_VEL
LIN {X 0,Y 394.034,Z 258.327,A -85,B 0,C 180,E1 -11818.788,E2 -11818.788} C_VEL
LIN {X 0,Y 396.231,Z 153.374,A -85,B 0,C 180,E1 -11820.732,E2 -11820.732} C_VEL
LIN {X 0,Y 393.199,Z 140.684,A -85,B 0,C 180,E1 -11821.214,E2 -11821.214} C_VEL
LIN {X 0,Y 386.081,Z 124.07,A -85,B 0,C 180,E1 -11822.113,E2 -11822.113} C_VEL
LIN {X 0,Y 383.317,Z 112.104,A -85,B 0,C 180,E1 -11825.278,E2 -11825.278} C_VEL
LIN {X 0,Y 383.006,Z 110.904,A -85,B 0,C 180,E1 -11825.634,E2 -11825.634} C_VEL
LIN {X 0,Y 382.979,Z 110.904,A -85,B 0,C 180,E1 -11828.604,E2 -11828.604} C_VEL
LIN {X 0,Y 382.961,Z 110.907,A -85,B 0,C 180,E1 -11831.351,E2 -11831.351} C_VEL
LIN {X 0,Y 382.99,Z 110.902,A -85,B 0,C 180,E1 -11834.302,E2 -11834.302} C_VEL
LIN {X 0,Y 382.997,Z 110.9,A -85,B 0,C 180,E1 -11837.238,E2 -11837.238} C_VEL
LIN {X 0,Y 382.986,Z 110.888,A -85,B 0,C 180,E1 -11840.419,E2 -11840.419} C_VEL
LIN {X 0,Y 383.015,Z 110.895,A -85,B 0,C 180,E1 -11844.043,E2 -11844.043} C_VEL
LIN {X 0,Y 382.987,Z 110.904,A -85,B 0,C 180,E1 -11847.578,E2 -11847.578} C_VEL
LIN {X 0,Y 382.979,Z 110.898,A -85,B 0,C 180,E1 -11850.299,E2 -11850.299} C_VEL
LIN {X 0,Y 383.005,Z 110.894,A -85,B 0,C 180,E1 -11854.044,E2 -11854.044} C_VEL
LIN {X 0,Y 382.99,Z 110.895,A -85,B 0,C 180,E1 -11857.334,E2 -11857.334} C_VEL
LIN {X 0,Y 383.059,Z 110.892,A -85,B 0,C 180,E1 -11860.716,E2 -11860.716} C_VEL
LIN {X 0,Y 383.081,Z 110.891,A -85,B 0,C 180,E1 -11864.026,E2 -11864.026} C_VEL
LIN {X 0,Y 383.137,Z 110.88,A -85,B 0,C 180,E1 -11867.284,E2 -11867.284} C_VEL
LIN {X 0,Y 383.144,Z 110.876,A -85,B 0,C 180,E1 -11870.498,E2 -11870.498} C_VEL
LIN {X 0,Y 383.264,Z 110.868,A -85,B 0,C 180,E1 -11873.683,E2 -11873.683} C_VEL
LIN {X 0,Y 383.384,Z 110.852,A -85,B 0,C 180,E1 -11877.899,E2 -11877.899} C_VEL
LIN {X 0,Y 383.516,Z 110.834,A -85,B 0,C 180,E1 -11880,E2 -11880} C_VEL
LIN {X 0,Y 383.239,Z 110.869,A -85,B 0,C 180,E1 -11883.154,E2 -11883.154} C_VEL
LIN {X 0,Y 383.243,Z 110.862,A -85,B 0,C 180,E1 -11886.317,E2 -11886.317} C_VEL
LIN {X 0,Y 383.144,Z 110.885,A -85,B 0,C 180,E1 -11889.502,E2 -11889.502} C_VEL
LIN {X 0,Y 383.126,Z 110.889,A -85,B 0,C 180,E1 -11893.536,E2 -11893.536} C_VEL
LIN {X 0,Y 383.096,Z 110.887,A -85,B 0,C 180,E1 -11897.455,E2 -11897.455} C_VEL
LIN {X 0,Y 383.029,Z 110.89,A -85,B 0,C 180,E1 -11900.647,E2 -11900.647} C_VEL
LIN {X 0,Y 383.034,Z 110.892,A -85,B 0,C 180,E1 -11903.807,E2 -11903.807} C_VEL
LIN {X 0,Y 383.081,Z 110.887,A -85,B 0,C 180,E1 -11906.123,E2 -11906.123} C_VEL
LIN {X 0,Y 383.041,Z 110.892,A -85,B 0,C 180,E1 -11908.493,E2 -11908.493} C_VEL
LIN {X 0,Y 383.01,Z 110.897,A -85,B 0,C 180,E1 -11912.15,E2 -11912.15} C_VEL
LIN {X 0,Y 383.018,Z 110.899,A -85,B 0,C 180,E1 -11914.668,E2 -11914.668} C_VEL
LIN {X 0,Y 382.998,Z 110.901,A -85,B 0,C 180,E1 -11917.903,E2 -11917.903} C_VEL
LIN {X 0,Y 382.984,Z 110.9,A -85,B 0,C 180,E1 -11921.347,E2 -11921.347} C_VEL
LIN {X 0,Y 382.996,Z 110.891,A -85,B 0,C 180,E1 -11924.303,E2 -11924.303} C_VEL
LIN {X 0,Y 383.01,Z 110.899,A -85,B 0,C 180,E1 -11927.24,E2 -11927.24} C_VEL
LIN {X 0,Y 383.016,Z 110.898,A -85,B 0,C 180,E1 -11930.413,E2 -11930.413} C_VEL
LIN {X 0,Y 383.026,Z 110.894,A -85,B 0,C 180,E1 -11934.044,E2 -11934.044} C_VEL
LIN {X 0,Y 383.018,Z 110.955,A -85,B 0,C 180,E1 -11937.405,E2 -11937.405} C_VEL
LIN {X 0,Y 386.248,Z 123.711,A -85,B 0,C 180,E1 -11940.575,E2 -11940.575} C_VEL
LIN {X 0,Y 388.591,Z 134.557,A -85,B 0,C 180,E1 -11943.118,E2 -11943.118} C_VEL
LIN {X 0,Y 388.793,Z 138.641,A -85,B 0,C 180,E1 -11944.002,E2 -11944.002} C_VEL
LIN {X 0,Y 388.694,Z 139.296,A -85,B 0,C 180,E1 -11944.133,E2 -11944.133} C_VEL
LIN {X 0,Y 394.999,Z 169.451,A -85,B 0,C 180,E1 -11945.225,E2 -11945.225} C_VEL
LIN {X 0,Y 395.847,Z 174.832,A -85,B 0,C 180,E1 -11945.395,E2 -11945.395} C_VEL
LIN {X 0,Y 393.744,Z 276.897,A -85,B 0,C 180,E1 -11947.295,E2 -11947.295} C_VEL
LIN {X 0,Y 392.947,Z 291.6,A -85,B 0,C 180,E1 -11947.766,E2 -11947.766} C_VEL
LIN {X 0,Y 391.851,Z 305.579,A -85,B 0,C 180,E1 -11948.428,E2 -11948.428} C_VEL
LIN {X 0,Y 390.656,Z 318.837,A -85,B 0,C 180,E1 -11949.278,E2 -11949.278} C_VEL
LIN {X 0,Y 389.282,Z 331.857,A -85,B 0,C 180,E1 -11950.351,E2 -11950.351} C_VEL
LIN {X 0,Y 387.801,Z 344.393,A -85,B 0,C 180,E1 -11951.646,E2 -11951.646} C_VEL
LIN {X 0,Y 386.345,Z 355.589,A -85,B 0,C 180,E1 -11953.079,E2 -11953.079} C_VEL
LIN {X 0,Y 385.032,Z 365.631,A -85,B 0,C 180,E1 -11954.653,E2 -11954.653} C_VEL
LIN {X 0,Y 384.01,Z 373.988,A -85,B 0,C 180,E1 -11956.236,E2 -11956.236} C_VEL
LIN {X 0,Y 383.233,Z 380.976,A -85,B 0,C 180,E1 -11957.825,E2 -11957.825} C_VEL
LIN {X 0,Y 382.52,Z 386.757,A -85,B 0,C 180,E1 -11959.413,E2 -11959.413} C_VEL
LIN {X 0,Y 382.112,Z 391.527,A -85,B 0,C 180,E1 -11961.006,E2 -11961.006} C_VEL
LIN {X 0,Y 381.737,Z 396.477,A -85,B 0,C 180,E1 -11963.127,E2 -11963.127} C_VEL
LIN {X 0,Y 381.608,Z 399.212,A -85,B 0,C 180,E1 -11964.716,E2 -11964.716} C_VEL
LIN {X 0,Y 381.514,Z 401.62,A -85,B 0,C 180,E1 -11966.832,E2 -11966.832} C_VEL
LIN {X 0,Y 381.571,Z 402.688,A -85,B 0,C 180,E1 -11968.944,E2 -11968.944} C_VEL
LIN {X 0,Y 381.588,Z 402.425,A -85,B 0,C 180,E1 -11971.055,E2 -11971.055} C_VEL
LIN {X 0,Y 381.531,Z 400.821,A -85,B 0,C 180,E1 -11973.168,E2 -11973.168} C_VEL
LIN {X 0,Y 381.589,Z 397.837,A -85,B 0,C 180,E1 -11975.284,E2 -11975.284} C_VEL
LIN {X 0,Y 381.765,Z 393.384,A -85,B 0,C 180,E1 -11977.404,E2 -11977.404} C_VEL
LIN {X 0,Y 381.994,Z 388.961,A -85,B 0,C 180,E1 -11978.997,E2 -11978.997} C_VEL
LIN {X 0,Y 382.476,Z 382.55,A -85,B 0,C 180,E1 -11980.856,E2 -11980.856} C_VEL
LIN {X 0,Y 383.172,Z 374.567,A -85,B 0,C 180,E1 -11982.715,E2 -11982.715} C_VEL
LIN {X 0,Y 383.888,Z 366.507,A -85,B 0,C 180,E1 -11984.255,E2 -11984.255} C_VEL
LIN {X 0,Y 384.979,Z 356.135,A -85,B 0,C 180,E1 -11985.892,E2 -11985.892} C_VEL
LIN {X 0,Y 386.068,Z 344.9,A -85,B 0,C 180,E1 -11987.343,E2 -11987.343} C_VEL
LIN {X 0,Y 387.194,Z 333.713,A -85,B 0,C 180,E1 -11988.52,E2 -11988.52} C_VEL
LIN {X 0,Y 388.343,Z 321.511,A -85,B 0,C 180,E1 -11989.562,E2 -11989.562} C_VEL
LIN {X 0,Y 389.406,Z 307.994,A -85,B 0,C 180,E1 -11990.467,E2 -11990.467} C_VEL
LIN {X 0,Y 390.273,Z 293.832,A -85,B 0,C 180,E1 -11991.179,E2 -11991.179} C_VEL
LIN {X 0,Y 390.964,Z 279.996,A -85,B 0,C 180,E1 -11991.658,E2 -11991.658} C_VEL
LIN {X 0,Y 391.444,Z 259.494,A -85,B 0,C 180,E1 -11992.08,E2 -11992.08} C_VEL
LIN {X 0,Y 392.801,Z 172.527,A -85,B 0,C 180,E1 -11993.674,E2 -11993.674} C_VEL
LIN {X 0,Y 387.036,Z 139.363,A -85,B 0,C 180,E1 -11994.686,E2 -11994.686} C_VEL
LIN {X 0,Y 387.597,Z 132.339,A -85,B 0,C 180,E1 -11996.085,E2 -11996.085} C_VEL
LIN {X 0,Y 385.61,Z 122.313,A -85,B 0,C 180,E1 -11998.285,E2 -11998.285} C_VEL
LIN {X 0,Y 383.009,Z 110.903,A -85,B 0,C 180,E1 -12000.916,E2 -12000.916} C_VEL
LIN {X 0,Y 383.017,Z 110.898,A -85,B 0,C 180,E1 -12004.668,E2 -12004.668} C_VEL
LIN {X 0,Y 382.998,Z 110.904,A -85,B 0,C 180,E1 -12007.903,E2 -12007.903} C_VEL
LIN {X 0,Y 382.983,Z 110.902,A -85,B 0,C 180,E1 -12011.347,E2 -12011.347} C_VEL
LIN {X 0,Y 383.008,Z 110.899,A -85,B 0,C 180,E1 -12014.305,E2 -12014.305} C_VEL
LIN {X 0,Y 383.074,Z 110.891,A -85,B 0,C 180,E1 -12017.249,E2 -12017.249} C_VEL
LIN {X 0,Y 383.015,Z 110.897,A -85,B 0,C 180,E1 -12020.413,E2 -12020.413} C_VEL
LIN {X 0,Y 383.023,Z 110.897,A -85,B 0,C 180,E1 -12024.044,E2 -12024.044} C_VEL
LIN {X 0,Y 382.985,Z 110.905,A -85,B 0,C 180,E1 -12027.578,E2 -12027.578} C_VEL
LIN {X 0,Y 382.991,Z 110.899,A -85,B 0,C 180,E1 -12030.3,E2 -12030.3} C_VEL
LIN {X 0,Y 383.055,Z 110.893,A -85,B 0,C 180,E1 -12032.698,E2 -12032.698} C_VEL
LIN {X 0,Y 383.032,Z 110.894,A -85,B 0,C 180,E1 -12036.193,E2 -12036.193} C_VEL
LIN {X 0,Y 383.054,Z 110.893,A -85,B 0,C 180,E1 -12039.599,E2 -12039.599} C_VEL
LIN {X 0,Y 383.104,Z 110.891,A -85,B 0,C 180,E1 -12042.931,E2 -12042.931} C_VEL
LIN {X 0,Y 383.124,Z 110.886,A -85,B 0,C 180,E1 -12046.464,E2 -12046.464} C_VEL
LIN {X 0,Y 383.15,Z 110.885,A -85,B 0,C 180,E1 -12050.498,E2 -12050.498} C_VEL
LIN {X 0,Y 383.28,Z 110.864,A -85,B 0,C 180,E1 -12053.684,E2 -12053.684} C_VEL
LIN {X 0,Y 383.384,Z 110.852,A -85,B 0,C 180,E1 -12057.899,E2 -12057.899} C_VEL
LIN {X 0,Y 383.517,Z 110.837,A -85,B 0,C 180,E1 -12060,E2 -12060} C_VEL
LIN {X 0,Y 383.246,Z 110.868,A -85,B 0,C 180,E1 -12063.154,E2 -12063.154} C_VEL
LIN {X 0,Y 383.245,Z 110.87,A -85,B 0,C 180,E1 -12066.494,E2 -12066.494} C_VEL
LIN {X 0,Y 383.15,Z 110.881,A -85,B 0,C 180,E1 -12069.502,E2 -12069.502} C_VEL
LIN {X 0,Y 383.125,Z 110.886,A -85,B 0,C 180,E1 -12073.536,E2 -12073.536} C_VEL
LIN {X 0,Y 383.094,Z 110.89,A -85,B 0,C 180,E1 -12077.455,E2 -12077.455} C_VEL
LIN {X 0,Y 383.031,Z 110.894,A -85,B 0,C 180,E1 -12080.648,E2 -12080.648} C_VEL
LIN {X 0,Y 383.033,Z 110.898,A -85,B 0,C 180,E1 -12083.808,E2 -12083.808} C_VEL
LIN {X 0,Y 383.079,Z 110.889,A -85,B 0,C 180,E1 -12086.124,E2 -12086.124} C_VEL
LIN {X 0,Y 382.992,Z 110.902,A -85,B 0,C 180,E1 -12089.7,E2 -12089.7} C_VEL
LIN {X 0,Y 383.003,Z 110.902,A -85,B 0,C 180,E1 -12093.401,E2 -12093.401} C_VEL
LIN {X 0,Y 383.031,Z 110.894,A -85,B 0,C 180,E1 -12096.165,E2 -12096.165} C_VEL
LIN {X 0,Y 383.008,Z 110.897,A -85,B 0,C 180,E1 -12099.959,E2 -12099.959} C_VEL
LIN {X 0,Y 383.006,Z 110.903,A -85,B 0,C 180,E1 -12102.779,E2 -12102.779} C_VEL
LIN {X 0,Y 382.997,Z 110.899,A -85,B 0,C 180,E1 -12105.79,E2 -12105.79} C_VEL
LIN {X 0,Y 382.987,Z 110.905,A -85,B 0,C 180,E1 -12108.797,E2 -12108.797} C_VEL
LIN {X 0,Y 382.998,Z 110.9,A -85,B 0,C 180,E1 -12112.097,E2 -12112.097} C_VEL
LIN {X 0,Y 383.019,Z 110.896,A -85,B 0,C 180,E1 -12115.333,E2 -12115.333} C_VEL
LIN {X 0,Y 382.984,Z 110.901,A -85,B 0,C 180,E1 -12119.082,E2 -12119.082} C_VEL
LIN {X 0,Y 382.995,Z 110.901,A -85,B 0,C 180,E1 -12122.694,E2 -12122.694} C_VEL
LIN {X 0,Y 383.017,Z 110.902,A -85,B 0,C 180,E1 -12126.192,E2 -12126.192} C_VEL
LIN {X 0,Y 383.046,Z 111.062,A -85,B 0,C 180,E1 -12128.19,E2 -12128.19} C_VEL
LIN {X 0,Y 385.803,Z 123.729,A -85,B 0,C 180,E1 -12131.31,E2 -12131.31} C_VEL
LIN {X 0,Y 390.045,Z 136.212,A -85,B 0,C 180,E1 -12131.835,E2 -12131.835} C_VEL
LIN {X 0,Y 393.124,Z 151.823,A -85,B 0,C 180,E1 -12132.319,E2 -12132.319} C_VEL
LIN {X 0,Y 391.298,Z 260.682,A -85,B 0,C 180,E1 -12134.338,E2 -12134.338} C_VEL
LIN {X 0,Y 390.785,Z 275.137,A -85,B 0,C 180,E1 -12134.818,E2 -12134.818} C_VEL
LIN {X 0,Y 389.942,Z 289.558,A -85,B 0,C 180,E1 -12135.518,E2 -12135.518} C_VEL
LIN {X 0,Y 388.94,Z 303.212,A -85,B 0,C 180,E1 -12136.414,E2 -12136.414} C_VEL
LIN {X 0,Y 387.905,Z 315.462,A -85,B 0,C 180,E1 -12137.443,E2 -12137.443} C_VEL
LIN {X 0,Y 386.878,Z 326.79,A -85,B 0,C 180,E1 -12138.619,E2 -12138.619} C_VEL
LIN {X 0,Y 385.683,Z 338.08,A -85,B 0,C 180,E1 -12140.046,E2 -12140.046} C_VEL
LIN {X 0,Y 384.624,Z 348.065,A -85,B 0,C 180,E1 -12141.595,E2 -12141.595} C_VEL
LIN {X 0,Y 383.833,Z 356.432,A -85,B 0,C 180,E1 -12143.165,E2 -12143.165} C_VEL
LIN {X 0,Y 382.964,Z 364.441,A -85,B 0,C 180,E1 -12144.999,E2 -12144.999} C_VEL
LIN {X 0,Y 382.285,Z 370.906,A -85,B 0,C 180,E1 -12146.839,E2 -12146.839} C_VEL
LIN {X 0,Y 381.871,Z 376.646,A -85,B 0,C 180,E1 -12148.946,E2 -12148.946} C_VEL
LIN {X 0,Y 381.717,Z 380.84,A -85,B 0,C 180,E1 -12151.055,E2 -12151.055} C_VEL
LIN {X 0,Y 381.564,Z 383.616,A -85,B 0,C 180,E1 -12153.168,E2 -12153.168} C_VEL
LIN {X 0,Y 381.587,Z 385.041,A -85,B 0,C 180,E1 -12155.284,E2 -12155.284} C_VEL
LIN {X 0,Y 381.628,Z 385.244,A -85,B 0,C 180,E1 -12156.255,E2 -12156.255} C_VEL
LIN {X 0,Y 380.867,Z 385.29,A -85,B 0,C 180,E1 -12157.136,E2 -12157.136} C_VEL
LIN {X 0,Y 377.964,Z 384.902,A -85,B 0,C 180,E1 -12158.567,E2 -12158.567} C_VEL
LIN {X 0,Y 375.599,Z 384.089,A -85,B 0,C 180,E1 -12159.717,E2 -12159.717} C_VEL
LIN {X 0,Y 374.641,Z 383.133,A -85,B 0,C 180,E1 -12160.599,E2 -12160.599} C_VEL
LIN {X 0,Y 374.591,Z 382.742,A -85,B 0,C 180,E1 -12160.896,E2 -12160.896} C_VEL
LIN {X 0,Y 374.984,Z 379.473,A -85,B 0,C 180,E1 -12162.997,E2 -12162.997} C_VEL
LIN {X 0,Y 375.468,Z 374.573,A -85,B 0,C 180,E1 -12165.192,E2 -12165.192} C_VEL
LIN {X 0,Y 376.048,Z 369.814,A -85,B 0,C 180,E1 -12166.839,E2 -12166.839} C_VEL
LIN {X 0,Y 376.976,Z 362.881,A -85,B 0,C 180,E1 -12168.759,E2 -12168.759} C_VEL
LIN {X 0,Y 378.152,Z 354.242,A -85,B 0,C 180,E1 -12170.678,E2 -12170.678} C_VEL
LIN {X 0,Y 379.546,Z 344.763,A -85,B 0,C 180,E1 -12172.382,E2 -12172.382} C_VEL
LIN {X 0,Y 380.903,Z 334.159,A -85,B 0,C 180,E1 -12173.949,E2 -12173.949} C_VEL
LIN {X 0,Y 382.484,Z 322.174,A -85,B 0,C 180,E1 -12175.376,E2 -12175.376} C_VEL
LIN {X 0,Y 383.838,Z 310.437,A -85,B 0,C 180,E1 -12176.507,E2 -12176.507} C_VEL
LIN {X 0,Y 385.129,Z 298.381,A -85,B 0,C 180,E1 -12177.437,E2 -12177.437} C_VEL
LIN {X 0,Y 386.192,Z 285.112,A -85,B 0,C 180,E1 -12178.239,E2 -12178.239} C_VEL
LIN {X 0,Y 387.066,Z 271.632,A -85,B 0,C 180,E1 -12178.836,E2 -12178.836} C_VEL
LIN {X 0,Y 387.631,Z 258.258,A -85,B 0,C 180,E1 -12179.235,E2 -12179.235} C_VEL
LIN {X 0,Y 389.908,Z 154.719,A -85,B 0,C 180,E1 -12181.181,E2 -12181.181} C_VEL
LIN {X 0,Y 387.173,Z 143.17,A -85,B 0,C 180,E1 -12181.63,E2 -12181.63} C_VEL
LIN {X 0,Y 379.972,Z 126.825,A -85,B 0,C 180,E1 -12182.556,E2 -12182.556} C_VEL
LIN {X 0,Y 378.869,Z 124.103,A -85,B 0,C 180,E1 -12182.739,E2 -12182.739} C_VEL
LIN {X 0,Y 376.306,Z 113.172,A -85,B 0,C 180,E1 -12185.707,E2 -12185.707} C_VEL
LIN {X 0,Y 375.987,Z 111.776,A -85,B 0,C 180,E1 -12186.125,E2 -12186.125} C_VEL
LIN {X 0,Y 375.933,Z 111.785,A -85,B 0,C 180,E1 -12189.466,E2 -12189.466} C_VEL
LIN {X 0,Y 375.934,Z 111.782,A -85,B 0,C 180,E1 -12193.189,E2 -12193.189} C_VEL
LIN {X 0,Y 375.933,Z 111.777,A -85,B 0,C 180,E1 -12196.811,E2 -12196.811} C_VEL
LIN {X 0,Y 375.935,Z 111.766,A -85,B 0,C 180,E1 -12200.534,E2 -12200.534} C_VEL
LIN {X 0,Y 375.959,Z 111.777,A -85,B 0,C 180,E1 -12203.497,E2 -12203.497} C_VEL
LIN {X 0,Y 375.958,Z 111.777,A -85,B 0,C 180,E1 -12205.888,E2 -12205.888} C_VEL
LIN {X 0,Y 375.963,Z 111.773,A -85,B 0,C 180,E1 -12209.687,E2 -12209.687} C_VEL
LIN {X 0,Y 375.929,Z 111.781,A -85,B 0,C 180,E1 -12212.136,E2 -12212.136} C_VEL
LIN {X 0,Y 375.969,Z 111.776,A -85,B 0,C 180,E1 -12215.717,E2 -12215.717} C_VEL
LIN {X 0,Y 375.999,Z 111.774,A -85,B 0,C 180,E1 -12219.198,E2 -12219.198} C_VEL
LIN {X 0,Y 376.033,Z 111.765,A -85,B 0,C 180,E1 -12222.6,E2 -12222.6} C_VEL
LIN {X 0,Y 376.091,Z 111.756,A -85,B 0,C 180,E1 -12226.342,E2 -12226.342} C_VEL
LIN {X 0,Y 376.114,Z 111.753,A -85,B 0,C 180,E1 -12230.318,E2 -12230.318} C_VEL
LIN {X 0,Y 376.22,Z 111.745,A -85,B 0,C 180,E1 -12233.564,E2 -12233.564} C_VEL
LIN {X 0,Y 376.35,Z 111.728,A -85,B 0,C 180,E1 -12237.859,E2 -12237.859} C_VEL
LIN {X 0,Y 376.486,Z 111.709,A -85,B 0,C 180,E1 -12240,E2 -12240} C_VEL
LIN {X 0,Y 376.349,Z 111.725,A -85,B 0,C 180,E1 -12242.14,E2 -12242.14} C_VEL
LIN {X 0,Y 376.201,Z 111.738,A -85,B 0,C 180,E1 -12246.436,E2 -12246.436} C_VEL
LIN {X 0,Y 376.114,Z 111.759,A -85,B 0,C 180,E1 -12249.681,E2 -12249.681} C_VEL
LIN {X 0,Y 376.09,Z 111.764,A -85,B 0,C 180,E1 -12253.657,E2 -12253.657} C_VEL
LIN {X 0,Y 376.044,Z 111.767,A -85,B 0,C 180,E1 -12257.607,E2 -12257.607} C_VEL
LIN {X 0,Y 375.979,Z 111.768,A -85,B 0,C 180,E1 -12260.832,E2 -12260.832} C_VEL
LIN {X 0,Y 375.995,Z 111.769,A -85,B 0,C 180,E1 -12264.281,E2 -12264.281} C_VEL
LIN {X 0,Y 376.02,Z 111.769,A -85,B 0,C 180,E1 -12266.652,E2 -12266.652} C_VEL
LIN {X 0,Y 375.971,Z 111.772,A -85,B 0,C 180,E1 -12269.079,E2 -12269.079} C_VEL
LIN {X 0,Y 375.95,Z 111.777,A -85,B 0,C 180,E1 -12272.828,E2 -12272.828} C_VEL
LIN {X 0,Y 375.958,Z 111.773,A -85,B 0,C 180,E1 -12275.415,E2 -12275.415} C_VEL
LIN {X 0,Y 375.973,Z 111.772,A -85,B 0,C 180,E1 -12278.27,E2 -12278.27} C_VEL
LIN {X 0,Y 375.935,Z 111.779,A -85,B 0,C 180,E1 -12281.601,E2 -12281.601} C_VEL
LIN {X 0,Y 375.927,Z 111.775,A -85,B 0,C 180,E1 -12285.269,E2 -12285.269} C_VEL
LIN {X 0,Y 375.935,Z 111.784,A -85,B 0,C 180,E1 -12288.399,E2 -12288.399} C_VEL
LIN {X 0,Y 375.975,Z 111.775,A -85,B 0,C 180,E1 -12291.729,E2 -12291.729} C_VEL
LIN {X 0,Y 375.98,Z 111.77,A -85,B 0,C 180,E1 -12295.333,E2 -12295.333} C_VEL
LIN {X 0,Y 375.981,Z 111.81,A -85,B 0,C 180,E1 -12296.895,E2 -12296.895} C_VEL
LIN {X 0,Y 378.981,Z 123.801,A -85,B 0,C 180,E1 -12299.954,E2 -12299.954} C_VEL
LIN {X 0,Y 381.451,Z 134.627,A -85,B 0,C 180,E1 -12302.573,E2 -12302.573} C_VEL
LIN {X 0,Y 382.078,Z 139.216,A -85,B 0,C 180,E1 -12303.607,E2 -12303.607} C_VEL
LIN {X 0,Y 387.976,Z 167.054,A -85,B 0,C 180,E1 -12304.65,E2 -12304.65} C_VEL
LIN {X 0,Y 389.423,Z 175.036,A -85,B 0,C 180,E1 -12304.923,E2 -12304.923} C_VEL
LIN {X 0,Y 387.317,Z 277.038,A -85,B 0,C 180,E1 -12306.861,E2 -12306.861} C_VEL
LIN {X 0,Y 386.474,Z 291.623,A -85,B 0,C 180,E1 -12307.338,E2 -12307.338} C_VEL
LIN {X 0,Y 385.429,Z 304.989,A -85,B 0,C 180,E1 -12307.979,E2 -12307.979} C_VEL
LIN {X 0,Y 384.28,Z 317.296,A -85,B 0,C 180,E1 -12308.765,E2 -12308.765} C_VEL
LIN {X 0,Y 382.97,Z 329.295,A -85,B 0,C 180,E1 -12309.734,E2 -12309.734} C_VEL
LIN {X 0,Y 381.492,Z 341.084,A -85,B 0,C 180,E1 -12310.913,E2 -12310.913} C_VEL
LIN {X 0,Y 380.065,Z 351.873,A -85,B 0,C 180,E1 -12312.235,E2 -12312.235} C_VEL
LIN {X 0,Y 378.591,Z 362.556,A -85,B 0,C 180,E1 -12313.832,E2 -12313.832} C_VEL
LIN {X 0,Y 377.417,Z 371.374,A -85,B 0,C 180,E1 -12315.436,E2 -12315.436} C_VEL
LIN {X 0,Y 376.4,Z 379.877,A -85,B 0,C 180,E1 -12317.327,E2 -12317.327} C_VEL
LIN {X 0,Y 375.495,Z 386.73,A -85,B 0,C 180,E1 -12319.212,E2 -12319.212} C_VEL
LIN {X 0,Y 375.053,Z 391.47,A -85,B 0,C 180,E1 -12320.835,E2 -12320.835} C_VEL
LIN {X 0,Y 374.664,Z 396.392,A -85,B 0,C 180,E1 -12322.996,E2 -12322.996} C_VEL
LIN {X 0,Y 374.521,Z 399.103,A -85,B 0,C 180,E1 -12324.616,E2 -12324.616} C_VEL
LIN {X 0,Y 374.43,Z 401.487,A -85,B 0,C 180,E1 -12326.772,E2 -12326.772} C_VEL
LIN {X 0,Y 374.471,Z 402.531,A -85,B 0,C 180,E1 -12328.924,E2 -12328.924} C_VEL
LIN {X 0,Y 374.488,Z 402.244,A -85,B 0,C 180,E1 -12331.075,E2 -12331.075} C_VEL
LIN {X 0,Y 374.445,Z 400.616,A -85,B 0,C 180,E1 -12333.228,E2 -12333.228} C_VEL
LIN {X 0,Y 374.504,Z 397.608,A -85,B 0,C 180,E1 -12335.384,E2 -12335.384} C_VEL
LIN {X 0,Y 374.683,Z 393.128,A -85,B 0,C 180,E1 -12337.545,E2 -12337.545} C_VEL
LIN {X 0,Y 374.93,Z 388.676,A -85,B 0,C 180,E1 -12339.168,E2 -12339.168} C_VEL
LIN {X 0,Y 375.436,Z 382.233,A -85,B 0,C 180,E1 -12341.062,E2 -12341.062} C_VEL
LIN {X 0,Y 376.201,Z 374.216,A -85,B 0,C 180,E1 -12342.954,E2 -12342.954} C_VEL
LIN {X 0,Y 376.998,Z 365.816,A -85,B 0,C 180,E1 -12344.576,E2 -12344.576} C_VEL
LIN {X 0,Y 378.087,Z 355.696,A -85,B 0,C 180,E1 -12346.19,E2 -12346.19} C_VEL
LIN {X 0,Y 379.27,Z 344.385,A -85,B 0,C 180,E1 -12347.664,E2 -12347.664} C_VEL
LIN {X 0,Y 380.44,Z 333.118,A -85,B 0,C 180,E1 -12348.861,E2 -12348.861} C_VEL
LIN {X 0,Y 381.662,Z 320.193,A -85,B 0,C 180,E1 -12349.966,E2 -12349.966} C_VEL
LIN {X 0,Y 382.671,Z 307.124,A -85,B 0,C 180,E1 -12350.844,E2 -12350.844} C_VEL
LIN {X 0,Y 383.631,Z 292.724,A -85,B 0,C 180,E1 -12351.564,E2 -12351.564} C_VEL
LIN {X 0,Y 384.344,Z 278.418,A -85,B 0,C 180,E1 -12352.051,E2 -12352.051} C_VEL
LIN {X 0,Y 385.159,Z 240.361,A -85,B 0,C 180,E1 -12352.789,E2 -12352.789} C_VEL
LIN {X 0,Y 386.164,Z 173.345,A -85,B 0,C 180,E1 -12354.043,E2 -12354.043} C_VEL
LIN {X 0,Y 380.219,Z 139.353,A -85,B 0,C 180,E1 -12355.08,E2 -12355.08} C_VEL
LIN {X 0,Y 380.63,Z 133.349,A -85,B 0,C 180,E1 -12356.304,E2 -12356.304} C_VEL
LIN {X 0,Y 378.262,Z 121.878,A -85,B 0,C 180,E1 -12358.886,E2 -12358.886} C_VEL
LIN {X 0,Y 375.966,Z 111.78,A -85,B 0,C 180,E1 -12361.274,E2 -12361.274} C_VEL
LIN {X 0,Y 375.979,Z 111.774,A -85,B 0,C 180,E1 -12364.667,E2 -12364.667} C_VEL
LIN {X 0,Y 375.973,Z 111.777,A -85,B 0,C 180,E1 -12368.27,E2 -12368.27} C_VEL
LIN {X 0,Y 375.933,Z 111.782,A -85,B 0,C 180,E1 -12371.601,E2 -12371.601} C_VEL
LIN {X 0,Y 375.98,Z 111.774,A -85,B 0,C 180,E1 -12375.26,E2 -12375.26} C_VEL
LIN {X 0,Y 375.987,Z 111.773,A -85,B 0,C 180,E1 -12378.39,E2 -12378.39} C_VEL
LIN {X 0,Y 375.961,Z 111.778,A -85,B 0,C 180,E1 -12381.911,E2 -12381.911} C_VEL
LIN {X 0,Y 375.978,Z 111.778,A -85,B 0,C 180,E1 -12385.333,E2 -12385.333} C_VEL
LIN {X 0,Y 375.956,Z 111.776,A -85,B 0,C 180,E1 -12388.438,E2 -12388.438} C_VEL
LIN {X 0,Y 375.995,Z 111.771,A -85,B 0,C 180,E1 -12392.141,E2 -12392.141} C_VEL
LIN {X 0,Y 376.005,Z 111.771,A -85,B 0,C 180,E1 -12394.539,E2 -12394.539} C_VEL
LIN {X 0,Y 375.962,Z 111.775,A -85,B 0,C 180,E1 -12398.046,E2 -12398.046} C_VEL
LIN {X 0,Y 376.008,Z 111.771,A -85,B 0,C 180,E1 -12401.473,E2 -12401.473} C_VEL
LIN {X 0,Y 376.057,Z 111.77,A -85,B 0,C 180,E1 -12404.833,E2 -12404.833} C_VEL
LIN {X 0,Y 376.049,Z 111.765,A -85,B 0,C 180,E1 -12408.137,E2 -12408.137} C_VEL
LIN {X 0,Y 376.218,Z 111.744,A -85,B 0,C 180,E1 -12411.919,E2 -12411.919} C_VEL
LIN {X 0,Y 376.168,Z 111.754,A -85,B 0,C 180,E1 -12414.64,E2 -12414.64} C_VEL
LIN {X 0,Y 376.35,Z 111.728,A -85,B 0,C 180,E1 -12417.86,E2 -12417.86} C_VEL
LIN {X 0,Y 376.486,Z 111.713,A -85,B 0,C 180,E1 -12420,E2 -12420} C_VEL
LIN {X 0,Y 376.184,Z 111.747,A -85,B 0,C 180,E1 -12423.213,E2 -12423.213} C_VEL
LIN {X 0,Y 376.214,Z 111.746,A -85,B 0,C 180,E1 -12426.477,E2 -12426.477} C_VEL
LIN {X 0,Y 376.118,Z 111.759,A -85,B 0,C 180,E1 -12429.682,E2 -12429.682} C_VEL
LIN {X 0,Y 376.089,Z 111.764,A -85,B 0,C 180,E1 -12433.658,E2 -12433.658} C_VEL
LIN {X 0,Y 376.042,Z 111.77,A -85,B 0,C 180,E1 -12437.607,E2 -12437.607} C_VEL
LIN {X 0,Y 375.978,Z 111.773,A -85,B 0,C 180,E1 -12440.832,E2 -12440.832} C_VEL
LIN {X 0,Y 375.993,Z 111.771,A -85,B 0,C 180,E1 -12444.282,E2 -12444.282} C_VEL
LIN {X 0,Y 376.019,Z 111.768,A -85,B 0,C 180,E1 -12446.652,E2 -12446.652} C_VEL
LIN {X 0,Y 375.964,Z 111.775,A -85,B 0,C 180,E1 -12450.313,E2 -12450.313} C_VEL
LIN {X 0,Y 375.96,Z 111.775,A -85,B 0,C 180,E1 -12454.112,E2 -12454.112} C_VEL
LIN {X 0,Y 375.953,Z 111.779,A -85,B 0,C 180,E1 -12456.742,E2 -12456.742} C_VEL
LIN {X 0,Y 375.988,Z 111.772,A -85,B 0,C 180,E1 -12459.971,E2 -12459.971} C_VEL
LIN {X 0,Y 375.93,Z 111.779,A -85,B 0,C 180,E1 -12463.766,E2 -12463.766} C_VEL
LIN {X 0,Y 375.935,Z 111.784,A -85,B 0,C 180,E1 -12466.811,E2 -12466.811} C_VEL
LIN {X 0,Y 375.958,Z 111.781,A -85,B 0,C 180,E1 -12470.537,E2 -12470.537} C_VEL
LIN {X 0,Y 375.964,Z 111.775,A -85,B 0,C 180,E1 -12473.496,E2 -12473.496} C_VEL
LIN {X 0,Y 375.961,Z 111.776,A -85,B 0,C 180,E1 -12475.889,E2 -12475.889} C_VEL
LIN {X 0,Y 375.964,Z 111.776,A -85,B 0,C 180,E1 -12479.688,E2 -12479.688} C_VEL
LIN {X 0,Y 375.937,Z 111.783,A -85,B 0,C 180,E1 -12482.137,E2 -12482.137} C_VEL
LIN {X 0,Y 375.974,Z 111.776,A -85,B 0,C 180,E1 -12485.717,E2 -12485.717} C_VEL
LIN {X 0,Y 375.977,Z 111.874,A -85,B 0,C 180,E1 -12487.83,E2 -12487.83} C_VEL
LIN {X 0,Y 378.615,Z 123.956,A -85,B 0,C 180,E1 -12490.874,E2 -12490.874} C_VEL
LIN {X 0,Y 383.686,Z 138.317,A -85,B 0,C 180,E1 -12491.49,E2 -12491.49} C_VEL
LIN {X 0,Y 386.579,Z 153.232,A -85,B 0,C 180,E1 -12491.961,E2 -12491.961} C_VEL
LIN {X 0,Y 384.632,Z 261.025,A -85,B 0,C 180,E1 -12493.991,E2 -12493.991} C_VEL
LIN {X 0,Y 384.08,Z 275.427,A -85,B 0,C 180,E1 -12494.478,E2 -12494.478} C_VEL
LIN {X 0,Y 383.219,Z 289.814,A -85,B 0,C 180,E1 -12495.191,E2 -12495.191} C_VEL
LIN {X 0,Y 382.219,Z 302.579,A -85,B 0,C 180,E1 -12496.035,E2 -12496.035} C_VEL
LIN {X 0,Y 381.161,Z 314.982,A -85,B 0,C 180,E1 -12497.082,E2 -12497.082} C_VEL
LIN {X 0,Y 380.093,Z 326.309,A -85,B 0,C 180,E1 -12498.265,E2 -12498.265} C_VEL
LIN {X 0,Y 378.982,Z 336.417,A -85,B 0,C 180,E1 -12499.539,E2 -12499.539} C_VEL
LIN {X 0,Y 378.108,Z 345.473,A -85,B 0,C 180,E1 -12500.91,E2 -12500.91} C_VEL
LIN {X 0,Y 377.063,Z 354.308,A -85,B 0,C 180,E1 -12502.503,E2 -12502.503} C_VEL
LIN {X 0,Y 376.107,Z 362.776,A -85,B 0,C 180,E1 -12504.37,E2 -12504.37} C_VEL
LIN {X 0,Y 375.416,Z 369.607,A -85,B 0,C 180,E1 -12506.243,E2 -12506.243} C_VEL
LIN {X 0,Y 374.978,Z 374.335,A -85,B 0,C 180,E1 -12507.852,E2 -12507.852} C_VEL
LIN {X 0,Y 374.7,Z 379.236,A -85,B 0,C 180,E1 -12510,E2 -12510} C_VEL
LIN {X 0,Y 374.522,Z 382.663,A -85,B 0,C 180,E1 -12512.151,E2 -12512.151} C_VEL
LIN {X 0,Y 374.519,Z 384.711,A -85,B 0,C 180,E1 -12514.305,E2 -12514.305} C_VEL
LIN {X 0,Y 374.53,Z 385.432,A -85,B 0,C 180,E1 -12516.465,E2 -12516.465} C_VEL
LIN {X 0,Y 374.422,Z 384.825,A -85,B 0,C 180,E1 -12518.636,E2 -12518.636} C_VEL
LIN {X 0,Y 374.591,Z 382.742,A -85,B 0,C 180,E1 -12520.896,E2 -12520.896} C_VEL
LIN {X 0,Y 374.039,Z 381.594,A -85,B 0,C 180,E1 -12521.777,E2 -12521.777} C_VEL
LIN {X 0,Y 371.427,Z 379.318,A -85,B 0,C 180,E1 -12523.21,E2 -12523.21} C_VEL
LIN {X 0,Y 369.274,Z 377.188,A -85,B 0,C 180,E1 -12524.351,E2 -12524.351} C_VEL
LIN {X 0,Y 368.477,Z 375.245,A -85,B 0,C 180,E1 -12525.213,E2 -12525.213} C_VEL
LIN {X 0,Y 368.482,Z 374.51,A -85,B 0,C 180,E1 -12525.499,E2 -12525.499} C_VEL
LIN {X 0,Y 369.126,Z 369.729,A -85,B 0,C 180,E1 -12527.164,E2 -12527.164} C_VEL
LIN {X 0,Y 370.129,Z 362.739,A -85,B 0,C 180,E1 -12529.12,E2 -12529.12} C_VEL
LIN {X 0,Y 371.361,Z 354.035,A -85,B 0,C 180,E1 -12531.074,E2 -12531.074} C_VEL
LIN {X 0,Y 372.733,Z 345.2,A -85,B 0,C 180,E1 -12532.686,E2 -12532.686} C_VEL
LIN {X 0,Y 373.989,Z 335.763,A -85,B 0,C 180,E1 -12534.125,E2 -12534.125} C_VEL
LIN {X 0,Y 375.525,Z 324.827,A -85,B 0,C 180,E1 -12535.496,E2 -12535.496} C_VEL
LIN {X 0,Y 377.039,Z 312.811,A -85,B 0,C 180,E1 -12536.724,E2 -12536.724} C_VEL
LIN {X 0,Y 378.304,Z 301.27,A -85,B 0,C 180,E1 -12537.674,E2 -12537.674} C_VEL
LIN {X 0,Y 379.506,Z 288.867,A -85,B 0,C 180,E1 -12538.481,E2 -12538.481} C_VEL
LIN {X 0,Y 380.451,Z 275.151,A -85,B 0,C 180,E1 -12539.158,E2 -12539.158} C_VEL
LIN {X 0,Y 381.163,Z 261.133,A -85,B 0,C 180,E1 -12539.629,E2 -12539.629} C_VEL
LIN {X 0,Y 383.553,Z 155.642,A -85,B 0,C 180,E1 -12541.659,E2 -12541.659} C_VEL
LIN {X 0,Y 381.356,Z 146.167,A -85,B 0,C 180,E1 -12542.033,E2 -12542.033} C_VEL
LIN {X 0,Y 373.233,Z 127.732,A -85,B 0,C 180,E1 -12543.111,E2 -12543.111} C_VEL
LIN {X 0,Y 371.773,Z 124.39,A -85,B 0,C 180,E1 -12543.321,E2 -12543.321} C_VEL
LIN {X 0,Y 369.331,Z 114.251,A -85,B 0,C 180,E1 -12546.15,E2 -12546.15} C_VEL
LIN {X 0,Y 368.912,Z 112.653,A -85,B 0,C 180,E1 -12546.616,E2 -12546.616} C_VEL
LIN {X 0,Y 368.885,Z 112.662,A -85,B 0,C 180,E1 -12550.374,E2 -12550.374} C_VEL
LIN {X 0,Y 368.88,Z 112.663,A -85,B 0,C 180,E1 -12553.615,E2 -12553.615} C_VEL
LIN {X 0,Y 368.884,Z 112.655,A -85,B 0,C 180,E1 -12556.695,E2 -12556.695} C_VEL
LIN {X 0,Y 368.885,Z 112.645,A -85,B 0,C 180,E1 -12559.648,E2 -12559.648} C_VEL
LIN {X 0,Y 368.897,Z 112.66,A -85,B 0,C 180,E1 -12563.145,E2 -12563.145} C_VEL
LIN {X 0,Y 368.896,Z 112.657,A -85,B 0,C 180,E1 -12566.462,E2 -12566.462} C_VEL
LIN {X 0,Y 368.931,Z 112.655,A -85,B 0,C 180,E1 -12569.046,E2 -12569.046} C_VEL
LIN {X 0,Y 368.868,Z 112.661,A -85,B 0,C 180,E1 -12572.789,E2 -12572.789} C_VEL
LIN {X 0,Y 368.947,Z 112.653,A -85,B 0,C 180,E1 -12576.42,E2 -12576.42} C_VEL
LIN {X 0,Y 368.937,Z 112.653,A -85,B 0,C 180,E1 -12579.947,E2 -12579.947} C_VEL
LIN {X 0,Y 368.969,Z 112.648,A -85,B 0,C 180,E1 -12583.398,E2 -12583.398} C_VEL
LIN {X 0,Y 369.059,Z 112.632,A -85,B 0,C 180,E1 -12586.79,E2 -12586.79} C_VEL
LIN {X 0,Y 369.064,Z 112.634,A -85,B 0,C 180,E1 -12590.131,E2 -12590.131} C_VEL
LIN {X 0,Y 369.179,Z 112.622,A -85,B 0,C 180,E1 -12593.441,E2 -12593.441} C_VEL
LIN {X 0,Y 369.315,Z 112.604,A -85,B 0,C 180,E1 -12597.819,E2 -12597.819} C_VEL
LIN {X 0,Y 369.456,Z 112.585,A -85,B 0,C 180,E1 -12600,E2 -12600} C_VEL
LIN {X 0,Y 369.314,Z 112.602,A -85,B 0,C 180,E1 -12602.181,E2 -12602.181} C_VEL
LIN {X 0,Y 369.162,Z 112.615,A -85,B 0,C 180,E1 -12606.559,E2 -12606.559} C_VEL
LIN {X 0,Y 369.064,Z 112.635,A -85,B 0,C 180,E1 -12609.868,E2 -12609.868} C_VEL
LIN {X 0,Y 369.038,Z 112.641,A -85,B 0,C 180,E1 -12613.772,E2 -12613.772} C_VEL
LIN {X 0,Y 369.002,Z 112.644,A -85,B 0,C 180,E1 -12617.768,E2 -12617.768} C_VEL
LIN {X 0,Y 368.93,Z 112.647,A -85,B 0,C 180,E1 -12621.22,E2 -12621.22} C_VEL
LIN {X 0,Y 368.959,Z 112.644,A -85,B 0,C 180,E1 -12624.775,E2 -12624.775} C_VEL
LIN {X 0,Y 368.969,Z 112.648,A -85,B 0,C 180,E1 -12627.203,E2 -12627.203} C_VEL
LIN {X 0,Y 368.919,Z 112.652,A -85,B 0,C 180,E1 -12629.69,E2 -12629.69} C_VEL
LIN {X 0,Y 368.897,Z 112.657,A -85,B 0,C 180,E1 -12633.043,E2 -12633.043} C_VEL
LIN {X 0,Y 368.917,Z 112.652,A -85,B 0,C 180,E1 -12636.197,E2 -12636.197} C_VEL
LIN {X 0,Y 368.901,Z 112.644,A -85,B 0,C 180,E1 -12638.953,E2 -12638.953} C_VEL
LIN {X 0,Y 368.882,Z 112.66,A -85,B 0,C 180,E1 -12642.009,E2 -12642.009} C_VEL
LIN {X 0,Y 368.88,Z 112.651,A -85,B 0,C 180,E1 -12645.176,E2 -12645.176} C_VEL
LIN {X 0,Y 368.884,Z 112.662,A -85,B 0,C 180,E1 -12648.178,E2 -12648.178} C_VEL
LIN {X 0,Y 368.91,Z 112.653,A -85,B 0,C 180,E1 -12651.36,E2 -12651.36} C_VEL
LIN {X 0,Y 368.937,Z 112.648,A -85,B 0,C 180,E1 -12655.146,E2 -12655.146} C_VEL
LIN {X 0,Y 368.946,Z 112.766,A -85,B 0,C 180,E1 -12656.385,E2 -12656.385} C_VEL
LIN {X 0,Y 372.049,Z 125.004,A -85,B 0,C 180,E1 -12659.592,E2 -12659.592} C_VEL
LIN {X 0,Y 374.467,Z 135.476,A -85,B 0,C 180,E1 -12662.19,E2 -12662.19} C_VEL
LIN {X 0,Y 375.121,Z 138.995,A -85,B 0,C 180,E1 -12663.022,E2 -12663.022} C_VEL
LIN {X 0,Y 376.706,Z 144.53,A -85,B 0,C 180,E1 -12663.275,E2 -12663.275} C_VEL
LIN {X 0,Y 382.229,Z 171.024,A -85,B 0,C 180,E1 -12664.284,E2 -12664.284} C_VEL
LIN {X 0,Y 383.15,Z 177.117,A -85,B 0,C 180,E1 -12664.483,E2 -12664.483} C_VEL
LIN {X 0,Y 380.913,Z 277.185,A -85,B 0,C 180,E1 -12666.413,E2 -12666.413} C_VEL
LIN {X 0,Y 380.003,Z 291.669,A -85,B 0,C 180,E1 -12666.894,E2 -12666.894} C_VEL
LIN {X 0,Y 378.875,Z 305.54,A -85,B 0,C 180,E1 -12667.578,E2 -12667.578} C_VEL
LIN {X 0,Y 377.701,Z 317.593,A -85,B 0,C 180,E1 -12668.368,E2 -12668.368} C_VEL
LIN {X 0,Y 376.137,Z 331,A -85,B 0,C 180,E1 -12669.492,E2 -12669.492} C_VEL
LIN {X 0,Y 374.638,Z 342.457,A -85,B 0,C 180,E1 -12670.693,E2 -12670.693} C_VEL
LIN {X 0,Y 373.052,Z 353.958,A -85,B 0,C 180,E1 -12672.173,E2 -12672.173} C_VEL
LIN {X 0,Y 371.499,Z 364.266,A -85,B 0,C 180,E1 -12673.797,E2 -12673.797} C_VEL
LIN {X 0,Y 370.283,Z 372.923,A -85,B 0,C 180,E1 -12675.463,E2 -12675.463} C_VEL
LIN {X 0,Y 369.288,Z 380.961,A -85,B 0,C 180,E1 -12677.358,E2 -12677.358} C_VEL
LIN {X 0,Y 368.475,Z 386.705,A -85,B 0,C 180,E1 -12679.004,E2 -12679.004} C_VEL
LIN {X 0,Y 367.996,Z 391.415,A -85,B 0,C 180,E1 -12680.657,E2 -12680.657} C_VEL
LIN {X 0,Y 367.59,Z 396.31,A -85,B 0,C 180,E1 -12682.861,E2 -12682.861} C_VEL
LIN {X 0,Y 367.439,Z 398.994,A -85,B 0,C 180,E1 -12684.512,E2 -12684.512} C_VEL
LIN {X 0,Y 367.349,Z 401.354,A -85,B 0,C 180,E1 -12686.71,E2 -12686.71} C_VEL
LIN {X 0,Y 367.371,Z 402.374,A -85,B 0,C 180,E1 -12688.904,E2 -12688.904} C_VEL
LIN {X 0,Y 367.388,Z 402.063,A -85,B 0,C 180,E1 -12691.096,E2 -12691.096} C_VEL
LIN {X 0,Y 367.362,Z 400.411,A -85,B 0,C 180,E1 -12693.29,E2 -12693.29} C_VEL
LIN {X 0,Y 367.422,Z 397.376,A -85,B 0,C 180,E1 -12695.488,E2 -12695.488} C_VEL
LIN {X 0,Y 367.624,Z 392.869,A -85,B 0,C 180,E1 -12697.69,E2 -12697.69} C_VEL
LIN {X 0,Y 367.882,Z 388.389,A -85,B 0,C 180,E1 -12699.345,E2 -12699.345} C_VEL
LIN {X 0,Y 368.423,Z 381.915,A -85,B 0,C 180,E1 -12701.275,E2 -12701.275} C_VEL
LIN {X 0,Y 369.241,Z 373.862,A -85,B 0,C 180,E1 -12703.203,E2 -12703.203} C_VEL
LIN {X 0,Y 370.028,Z 365.419,A -85,B 0,C 180,E1 -12704.857,E2 -12704.857} C_VEL
LIN {X 0,Y 371.175,Z 355.25,A -85,B 0,C 180,E1 -12706.5,E2 -12706.5} C_VEL
LIN {X 0,Y 372.478,Z 343.855,A -85,B 0,C 180,E1 -12707.997,E2 -12707.997} C_VEL
LIN {X 0,Y 373.698,Z 332.508,A -85,B 0,C 180,E1 -12709.215,E2 -12709.215} C_VEL
LIN {X 0,Y 374.932,Z 319.471,A -85,B 0,C 180,E1 -12710.34,E2 -12710.34} C_VEL
LIN {X 0,Y 375.96,Z 306.244,A -85,B 0,C 180,E1 -12711.234,E2 -12711.234} C_VEL
LIN {X 0,Y 376.954,Z 292.37,A -85,B 0,C 180,E1 -12711.929,E2 -12711.929} C_VEL
LIN {X 0,Y 377.696,Z 277.968,A -85,B 0,C 180,E1 -12712.424,E2 -12712.424} C_VEL
LIN {X 0,Y 378.784,Z 221.865,A -85,B 0,C 180,E1 -12713.516,E2 -12713.516} C_VEL
LIN {X 0,Y 379.585,Z 174.32,A -85,B 0,C 180,E1 -12714.418,E2 -12714.418} C_VEL
LIN {X 0,Y 373.468,Z 139.181,A -85,B 0,C 180,E1 -12715.517,E2 -12715.517} C_VEL
LIN {X 0,Y 373.786,Z 135.766,A -85,B 0,C 180,E1 -12716.222,E2 -12716.222} C_VEL
LIN {X 0,Y 372.196,Z 127.195,A -85,B 0,C 180,E1 -12718.168,E2 -12718.168} C_VEL
LIN {X 0,Y 369.396,Z 114.763,A -85,B 0,C 180,E1 -12721.113,E2 -12721.113} C_VEL
LIN {X 0,Y 368.942,Z 112.655,A -85,B 0,C 180,E1 -12721.67,E2 -12721.67} C_VEL
LIN {X 0,Y 368.928,Z 112.651,A -85,B 0,C 180,E1 -12725.001,E2 -12725.001} C_VEL
LIN {X 0,Y 368.907,Z 112.655,A -85,B 0,C 180,E1 -12728.64,E2 -12728.64} C_VEL
LIN {X 0,Y 368.881,Z 112.662,A -85,B 0,C 180,E1 -12732.009,E2 -12732.009} C_VEL
LIN {X 0,Y 368.954,Z 112.649,A -85,B 0,C 180,E1 -12735.187,E2 -12735.187} C_VEL
LIN {X 0,Y 368.943,Z 112.651,A -85,B 0,C 180,E1 -12738.186,E2 -12738.186} C_VEL
LIN {X 0,Y 368.906,Z 112.658,A -85,B 0,C 180,E1 -12741.36,E2 -12741.36} C_VEL
LIN {X 0,Y 368.935,Z 112.653,A -85,B 0,C 180,E1 -12745.146,E2 -12745.146} C_VEL
LIN {X 0,Y 368.928,Z 112.655,A -85,B 0,C 180,E1 -12749.046,E2 -12749.046} C_VEL
LIN {X 0,Y 368.978,Z 112.648,A -85,B 0,C 180,E1 -12751.564,E2 -12751.564} C_VEL
LIN {X 0,Y 368.999,Z 112.643,A -85,B 0,C 180,E1 -12754.02,E2 -12754.02} C_VEL
LIN {X 0,Y 368.931,Z 112.652,A -85,B 0,C 180,E1 -12757.605,E2 -12757.605} C_VEL
LIN {X 0,Y 368.957,Z 112.652,A -85,B 0,C 180,E1 -12761.106,E2 -12761.106} C_VEL
LIN {X 0,Y 368.996,Z 112.646,A -85,B 0,C 180,E1 -12764.535,E2 -12764.535} C_VEL
LIN {X 0,Y 369.004,Z 112.642,A -85,B 0,C 180,E1 -12767.907,E2 -12767.907} C_VEL
LIN {X 0,Y 369.165,Z 112.622,A -85,B 0,C 180,E1 -12771.869,E2 -12771.869} C_VEL
LIN {X 0,Y 369.141,Z 112.631,A -85,B 0,C 180,E1 -12774.538,E2 -12774.538} C_VEL
LIN {X 0,Y 369.315,Z 112.604,A -85,B 0,C 180,E1 -12777.819,E2 -12777.819} C_VEL
LIN {X 0,Y 369.456,Z 112.589,A -85,B 0,C 180,E1 -12780,E2 -12780} C_VEL
LIN {X 0,Y 369.316,Z 112.609,A -85,B 0,C 180,E1 -12782.181,E2 -12782.181} C_VEL
LIN {X 0,Y 369.177,Z 112.622,A -85,B 0,C 180,E1 -12786.559,E2 -12786.559} C_VEL
LIN {X 0,Y 369.066,Z 112.639,A -85,B 0,C 180,E1 -12789.869,E2 -12789.869} C_VEL
LIN {X 0,Y 369.036,Z 112.643,A -85,B 0,C 180,E1 -12793.773,E2 -12793.773} C_VEL
LIN {X 0,Y 369,Z 112.648,A -85,B 0,C 180,E1 -12797.769,E2 -12797.769} C_VEL
LIN {X 0,Y 368.929,Z 112.654,A -85,B 0,C 180,E1 -12801.22,E2 -12801.22} C_VEL
LIN {X 0,Y 368.957,Z 112.648,A -85,B 0,C 180,E1 -12804.776,E2 -12804.776} C_VEL
LIN {X 0,Y 368.962,Z 112.651,A -85,B 0,C 180,E1 -12807.204,E2 -12807.204} C_VEL
LIN {X 0,Y 368.929,Z 112.654,A -85,B 0,C 180,E1 -12810.954,E2 -12810.954} C_VEL
LIN {X 0,Y 368.929,Z 112.656,A -85,B 0,C 180,E1 -12815.002,E2 -12815.002} C_VEL
LIN {X 0,Y 368.907,Z 112.656,A -85,B 0,C 180,E1 -12818.64,E2 -12818.64} C_VEL
LIN {X 0,Y 368.881,Z 112.657,A -85,B 0,C 180,E1 -12822.01,E2 -12822.01} C_VEL
LIN {X 0,Y 368.884,Z 112.659,A -85,B 0,C 180,E1 -12825.177,E2 -12825.177} C_VEL
LIN {X 0,Y 368.882,Z 112.658,A -85,B 0,C 180,E1 -12828.178,E2 -12828.178} C_VEL
LIN {X 0,Y 368.905,Z 112.655,A -85,B 0,C 180,E1 -12831.361,E2 -12831.361} C_VEL
LIN {X 0,Y 368.938,Z 112.651,A -85,B 0,C 180,E1 -12835.147,E2 -12835.147} C_VEL
LIN {X 0,Y 368.931,Z 112.652,A -85,B 0,C 180,E1 -12839.047,E2 -12839.047} C_VEL
LIN {X 0,Y 368.874,Z 112.659,A -85,B 0,C 180,E1 -12842.79,E2 -12842.79} C_VEL
LIN {X 0,Y 368.951,Z 112.652,A -85,B 0,C 180,E1 -12846.421,E2 -12846.421} C_VEL
LIN {X 0,Y 368.93,Z 112.676,A -85,B 0,C 180,E1 -12847.457,E2 -12847.457} C_VEL
LIN {X 0,Y 371.457,Z 124.152,A -85,B 0,C 180,E1 -12850.413,E2 -12850.413} C_VEL
LIN {X 0,Y 377.284,Z 140.229,A -85,B 0,C 180,E1 -12851.126,E2 -12851.126} C_VEL
LIN {X 0,Y 380.004,Z 154.467,A -85,B 0,C 180,E1 -12851.585,E2 -12851.585} C_VEL
LIN {X 0,Y 377.969,Z 261.356,A -85,B 0,C 180,E1 -12853.632,E2 -12853.632} C_VEL
LIN {X 0,Y 377.388,Z 275.704,A -85,B 0,C 180,E1 -12854.126,E2 -12854.126} C_VEL
LIN {X 0,Y 376.509,Z 290.061,A -85,B 0,C 180,E1 -12854.851,E2 -12854.851} C_VEL
LIN {X 0,Y 375.389,Z 303.687,A -85,B 0,C 180,E1 -12855.776,E2 -12855.776} C_VEL
LIN {X 0,Y 374.289,Z 315.908,A -85,B 0,C 180,E1 -12856.84,E2 -12856.84} C_VEL
LIN {X 0,Y 373.182,Z 327.101,A -85,B 0,C 180,E1 -12858.044,E2 -12858.044} C_VEL
LIN {X 0,Y 372.012,Z 337.336,A -85,B 0,C 180,E1 -12859.374,E2 -12859.374} C_VEL
LIN {X 0,Y 370.866,Z 347.692,A -85,B 0,C 180,E1 -12861.006,E2 -12861.006} C_VEL
LIN {X 0,Y 369.966,Z 356.173,A -85,B 0,C 180,E1 -12862.633,E2 -12862.633} C_VEL
LIN {X 0,Y 368.979,Z 364.314,A -85,B 0,C 180,E1 -12864.535,E2 -12864.535} C_VEL
LIN {X 0,Y 368.354,Z 370.014,A -85,B 0,C 180,E1 -12866.171,E2 -12866.171} C_VEL
LIN {X 0,Y 367.911,Z 374.691,A -85,B 0,C 180,E1 -12867.811,E2 -12867.811} C_VEL
LIN {X 0,Y 367.628,Z 379.542,A -85,B 0,C 180,E1 -12870,E2 -12870} C_VEL
LIN {X 0,Y 367.421,Z 382.925,A -85,B 0,C 180,E1 -12872.193,E2 -12872.193} C_VEL
LIN {X 0,Y 367.424,Z 384.929,A -85,B 0,C 180,E1 -12874.388,E2 -12874.388} C_VEL
LIN {X 0,Y 367.428,Z 385.6,A -85,B 0,C 180,E1 -12876.59,E2 -12876.59} C_VEL
LIN {X 0,Y 367.351,Z 384.938,A -85,B 0,C 180,E1 -12878.804,E2 -12878.804} C_VEL
LIN {X 0,Y 367.523,Z 382.919,A -85,B 0,C 180,E1 -12881.025,E2 -12881.025} C_VEL
LIN {X 0,Y 367.96,Z 379.491,A -85,B 0,C 180,E1 -12883.25,E2 -12883.25} C_VEL
LIN {X 0,Y 368.482,Z 374.51,A -85,B 0,C 180,E1 -12885.499,E2 -12885.499} C_VEL
LIN {X 0,Y 368.111,Z 372.29,A -85,B 0,C 180,E1 -12886.348,E2 -12886.348} C_VEL
LIN {X 0,Y 365.838,Z 368.403,A -85,B 0,C 180,E1 -12887.73,E2 -12887.73} C_VEL
LIN {X 0,Y 363.68,Z 364.077,A -85,B 0,C 180,E1 -12889.091,E2 -12889.091} C_VEL
LIN {X 0,Y 363.491,Z 361.022,A -85,B 0,C 180,E1 -12889.891,E2 -12889.891} C_VEL
LIN {X 0,Y 364.875,Z 352.446,A -85,B 0,C 180,E1 -12891.764,E2 -12891.764} C_VEL
LIN {X 0,Y 366.323,Z 343.091,A -85,B 0,C 180,E1 -12893.429,E2 -12893.429} C_VEL
LIN {X 0,Y 367.875,Z 332.308,A -85,B 0,C 180,E1 -12895.004,E2 -12895.004} C_VEL
LIN {X 0,Y 369.484,Z 321.068,A -85,B 0,C 180,E1 -12896.34,E2 -12896.34} C_VEL
LIN {X 0,Y 370.922,Z 309.046,A -85,B 0,C 180,E1 -12897.506,E2 -12897.506} C_VEL
LIN {X 0,Y 372.42,Z 296.566,A -85,B 0,C 180,E1 -12898.457,E2 -12898.457} C_VEL
LIN {X 0,Y 373.448,Z 283.95,A -85,B 0,C 180,E1 -12899.217,E2 -12899.217} C_VEL
LIN {X 0,Y 374.376,Z 270.057,A -85,B 0,C 180,E1 -12899.825,E2 -12899.825} C_VEL
LIN {X 0,Y 375.015,Z 255.719,A -85,B 0,C 180,E1 -12900.228,E2 -12900.228} C_VEL
LIN {X 0,Y 377.211,Z 156.362,A -85,B 0,C 180,E1 -12902.158,E2 -12902.158} C_VEL
LIN {X 0,Y 375.421,Z 148.912,A -85,B 0,C 180,E1 -12902.467,E2 -12902.467} C_VEL
LIN {X 0,Y 367.738,Z 131.453,A -85,B 0,C 180,E1 -12903.516,E2 -12903.516} C_VEL
LIN {X 0,Y 364.548,Z 124.487,A -85,B 0,C 180,E1 -12903.992,E2 -12903.992} C_VEL
LIN {X 0,Y 361.851,Z 113.532,A -85,B 0,C 180,E1 -12907.169,E2 -12907.169} C_VEL
LIN {X 0,Y 361.811,Z 113.542,A -85,B 0,C 180,E1 -12910.75,E2 -12910.75} C_VEL
LIN {X 0,Y 361.813,Z 113.54,A -85,B 0,C 180,E1 -12914.369,E2 -12914.369} C_VEL
LIN {X 0,Y 361.827,Z 113.541,A -85,B 0,C 180,E1 -12917.57,E2 -12917.57} C_VEL
LIN {X 0,Y 361.843,Z 113.531,A -85,B 0,C 180,E1 -12921.572,E2 -12921.572} C_VEL
LIN {X 0,Y 361.871,Z 113.53,A -85,B 0,C 180,E1 -12924.656,E2 -12924.656} C_VEL
LIN {X 0,Y 361.839,Z 113.537,A -85,B 0,C 180,E1 -12928.37,E2 -12928.37} C_VEL
LIN {X 0,Y 361.867,Z 113.531,A -85,B 0,C 180,E1 -12930.952,E2 -12930.952} C_VEL
LIN {X 0,Y 361.882,Z 113.529,A -85,B 0,C 180,E1 -12934.706,E2 -12934.706} C_VEL
LIN {X 0,Y 361.855,Z 113.529,A -85,B 0,C 180,E1 -12938.344,E2 -12938.344} C_VEL
LIN {X 0,Y 361.921,Z 113.519,A -85,B 0,C 180,E1 -12942.085,E2 -12942.085} C_VEL
LIN {X 0,Y 361.963,Z 113.517,A -85,B 0,C 180,E1 -12945.379,E2 -12945.379} C_VEL
LIN {X 0,Y 361.972,Z 113.521,A -85,B 0,C 180,E1 -12948.804,E2 -12948.804} C_VEL
LIN {X 0,Y 362.08,Z 113.501,A -85,B 0,C 180,E1 -12952.191,E2 -12952.191} C_VEL
LIN {X 0,Y 362.107,Z 113.502,A -85,B 0,C 180,E1 -12954.431,E2 -12954.431} C_VEL
LIN {X 0,Y 362.279,Z 113.48,A -85,B 0,C 180,E1 -12957.776,E2 -12957.776} C_VEL
LIN {X 0,Y 362.425,Z 113.46,A -85,B 0,C 180,E1 -12960,E2 -12960} C_VEL
LIN {X 0,Y 362.278,Z 113.478,A -85,B 0,C 180,E1 -12962.223,E2 -12962.223} C_VEL
LIN {X 0,Y 362.125,Z 113.491,A -85,B 0,C 180,E1 -12966.687,E2 -12966.687} C_VEL
LIN {X 0,Y 362.001,Z 113.513,A -85,B 0,C 180,E1 -12970.063,E2 -12970.063} C_VEL
LIN {X 0,Y 361.999,Z 113.517,A -85,B 0,C 180,E1 -12973.899,E2 -12973.899} C_VEL
LIN {X 0,Y 361.968,Z 113.519,A -85,B 0,C 180,E1 -12977.938,E2 -12977.938} C_VEL
LIN {X 0,Y 361.893,Z 113.527,A -85,B 0,C 180,E1 -12981.653,E2 -12981.653} C_VEL
LIN {X 0,Y 361.929,Z 113.519,A -85,B 0,C 180,E1 -12985.29,E2 -12985.29} C_VEL
LIN {X 0,Y 361.919,Z 113.523,A -85,B 0,C 180,E1 -12987.778,E2 -12987.778} C_VEL
LIN {X 0,Y 361.847,Z 113.534,A -85,B 0,C 180,E1 -12991.285,E2 -12991.285} C_VEL
LIN {X 0,Y 361.855,Z 113.537,A -85,B 0,C 180,E1 -12994.28,E2 -12994.28} C_VEL
LIN {X 0,Y 361.863,Z 113.534,A -85,B 0,C 180,E1 -12997.223,E2 -12997.223} C_VEL
LIN {X 0,Y 361.835,Z 113.526,A -85,B 0,C 180,E1 -13000.755,E2 -13000.755} C_VEL
LIN {X 0,Y 361.817,Z 113.528,A -85,B 0,C 180,E1 -13004.368,E2 -13004.368} C_VEL
LIN {X 0,Y 361.837,Z 113.537,A -85,B 0,C 180,E1 -13007.568,E2 -13007.568} C_VEL
LIN {X 0,Y 361.871,Z 113.529,A -85,B 0,C 180,E1 -13010.973,E2 -13010.973} C_VEL
LIN {X 0,Y 361.875,Z 113.529,A -85,B 0,C 180,E1 -13014.655,E2 -13014.655} C_VEL
LIN {X 0,Y 361.912,Z 113.689,A -85,B 0,C 180,E1 -13015.843,E2 -13015.843} C_VEL
LIN {X 0,Y 365.221,Z 126.688,A -85,B 0,C 180,E1 -13019.34,E2 -13019.34} C_VEL
LIN {X 0,Y 367.815,Z 138.163,A -85,B 0,C 180,E1 -13022.241,E2 -13022.241} C_VEL
LIN {X 0,Y 368.067,Z 139.176,A -85,B 0,C 180,E1 -13022.412,E2 -13022.412} C_VEL
LIN {X 0,Y 370.437,Z 145.488,A -85,B 0,C 180,E1 -13022.759,E2 -13022.759} C_VEL
LIN {X 0,Y 375.73,Z 171.093,A -85,B 0,C 180,E1 -13023.761,E2 -13023.761} C_VEL
LIN {X 0,Y 376.831,Z 177.281,A -85,B 0,C 180,E1 -13023.982,E2 -13023.982} C_VEL
LIN {X 0,Y 374.535,Z 277.345,A -85,B 0,C 180,E1 -13025.949,E2 -13025.949} C_VEL
LIN {X 0,Y 373.582,Z 291.722,A -85,B 0,C 180,E1 -13026.436,E2 -13026.436} C_VEL
LIN {X 0,Y 372.487,Z 304.972,A -85,B 0,C 180,E1 -13027.098,E2 -13027.098} C_VEL
LIN {X 0,Y 371.26,Z 316.771,A -85,B 0,C 180,E1 -13027.872,E2 -13027.872} C_VEL
LIN {X 0,Y 369.718,Z 329.869,A -85,B 0,C 180,E1 -13028.974,E2 -13028.974} C_VEL
LIN {X 0,Y 367.943,Z 342.666,A -85,B 0,C 180,E1 -13030.327,E2 -13030.327} C_VEL
LIN {X 0,Y 366.542,Z 352.16,A -85,B 0,C 180,E1 -13031.556,E2 -13031.556} C_VEL
LIN {X 0,Y 364.933,Z 362.74,A -85,B 0,C 180,E1 -13033.209,E2 -13033.209} C_VEL
LIN {X 0,Y 363.623,Z 371.492,A -85,B 0,C 180,E1 -13034.876,E2 -13034.876} C_VEL
LIN {X 0,Y 362.611,Z 378.781,A -85,B 0,C 180,E1 -13036.551,E2 -13036.551} C_VEL
LIN {X 0,Y 361.736,Z 384.871,A -85,B 0,C 180,E1 -13038.229,E2 -13038.229} C_VEL
LIN {X 0,Y 360.954,Z 391.362,A -85,B 0,C 180,E1 -13040.474,E2 -13040.474} C_VEL
LIN {X 0,Y 360.508,Z 396.228,A -85,B 0,C 180,E1 -13042.72,E2 -13042.72} C_VEL
LIN {X 0,Y 360.347,Z 398.887,A -85,B 0,C 180,E1 -13044.404,E2 -13044.404} C_VEL
LIN {X 0,Y 360.269,Z 401.222,A -85,B 0,C 180,E1 -13046.645,E2 -13046.645} C_VEL
LIN {X 0,Y 360.271,Z 402.217,A -85,B 0,C 180,E1 -13048.882,E2 -13048.882} C_VEL
LIN {X 0,Y 360.288,Z 401.881,A -85,B 0,C 180,E1 -13051.118,E2 -13051.118} C_VEL
LIN {X 0,Y 360.281,Z 400.205,A -85,B 0,C 180,E1 -13053.355,E2 -13053.355} C_VEL
LIN {X 0,Y 360.325,Z 397.144,A -85,B 0,C 180,E1 -13055.596,E2 -13055.596} C_VEL
LIN {X 0,Y 360.541,Z 392.608,A -85,B 0,C 180,E1 -13057.842,E2 -13057.842} C_VEL
LIN {X 0,Y 360.848,Z 388.1,A -85,B 0,C 180,E1 -13059.529,E2 -13059.529} C_VEL
LIN {X 0,Y 361.426,Z 381.593,A -85,B 0,C 180,E1 -13061.497,E2 -13061.497} C_VEL
LIN {X 0,Y 362.27,Z 373.504,A -85,B 0,C 180,E1 -13063.462,E2 -13063.462} C_VEL
LIN {X 0,Y 363.088,Z 365.02,A -85,B 0,C 180,E1 -13065.148,E2 -13065.148} C_VEL
LIN {X 0,Y 364.306,Z 354.795,A -85,B 0,C 180,E1 -13066.82,E2 -13066.82} C_VEL
LIN {X 0,Y 365.55,Z 344.491,A -85,B 0,C 180,E1 -13068.205,E2 -13068.205} C_VEL
LIN {X 0,Y 366.804,Z 333.318,A -85,B 0,C 180,E1 -13069.445,E2 -13069.445} C_VEL
LIN {X 0,Y 368.098,Z 320.138,A -85,B 0,C 180,E1 -13070.621,E2 -13070.621} C_VEL
LIN {X 0,Y 369.227,Z 306.497,A -85,B 0,C 180,E1 -13071.568,E2 -13071.568} C_VEL
LIN {X 0,Y 370.305,Z 291.999,A -85,B 0,C 180,E1 -13072.307,E2 -13072.307} C_VEL
LIN {X 0,Y 371.071,Z 277.494,A -85,B 0,C 180,E1 -13072.81,E2 -13072.81} C_VEL
LIN {X 0,Y 373.095,Z 176.429,A -85,B 0,C 180,E1 -13074.778,E2 -13074.778} C_VEL
LIN {X 0,Y 367.413,Z 143.003,A -85,B 0,C 180,E1 -13075.838,E2 -13075.838} C_VEL
LIN {X 0,Y 366.751,Z 138.865,A -85,B 0,C 180,E1 -13076.002,E2 -13076.002} C_VEL
LIN {X 0,Y 366.635,Z 135.347,A -85,B 0,C 180,E1 -13076.774,E2 -13076.774} C_VEL
LIN {X 0,Y 363.92,Z 122.455,A -85,B 0,C 180,E1 -13079.817,E2 -13079.817} C_VEL
LIN {X 0,Y 361.881,Z 113.535,A -85,B 0,C 180,E1 -13082.034,E2 -13082.034} C_VEL
LIN {X 0,Y 361.867,Z 113.534,A -85,B 0,C 180,E1 -13085.636,E2 -13085.636} C_VEL
LIN {X 0,Y 361.868,Z 113.531,A -85,B 0,C 180,E1 -13089.026,E2 -13089.026} C_VEL
LIN {X 0,Y 361.837,Z 113.535,A -85,B 0,C 180,E1 -13092.828,E2 -13092.828} C_VEL
LIN {X 0,Y 361.911,Z 113.53,A -85,B 0,C 180,E1 -13095.931,E2 -13095.931} C_VEL
LIN {X 0,Y 361.905,Z 113.528,A -85,B 0,C 180,E1 -13099.232,E2 -13099.232} C_VEL
LIN {X 0,Y 361.865,Z 113.532,A -85,B 0,C 180,E1 -13102.982,E2 -13102.982} C_VEL
LIN {X 0,Y 361.857,Z 113.532,A -85,B 0,C 180,E1 -13106.631,E2 -13106.631} C_VEL
LIN {X 0,Y 361.873,Z 113.533,A -85,B 0,C 180,E1 -13109.672,E2 -13109.672} C_VEL
LIN {X 0,Y 361.953,Z 113.523,A -85,B 0,C 180,E1 -13113.475,E2 -13113.475} C_VEL
LIN {X 0,Y 361.889,Z 113.534,A -85,B 0,C 180,E1 -13117.145,E2 -13117.145} C_VEL
LIN {X 0,Y 361.905,Z 113.53,A -85,B 0,C 180,E1 -13120.723,E2 -13120.723} C_VEL
LIN {X 0,Y 361.932,Z 113.527,A -85,B 0,C 180,E1 -13123.066,E2 -13123.066} C_VEL
LIN {X 0,Y 361.998,Z 113.518,A -85,B 0,C 180,E1 -13126.528,E2 -13126.528} C_VEL
LIN {X 0,Y 362.03,Z 113.511,A -85,B 0,C 180,E1 -13129.938,E2 -13129.938} C_VEL
LIN {X 0,Y 362.16,Z 113.494,A -85,B 0,C 180,E1 -13133.314,E2 -13133.314} C_VEL
LIN {X 0,Y 362.279,Z 113.481,A -85,B 0,C 180,E1 -13137.777,E2 -13137.777} C_VEL
LIN {X 0,Y 362.425,Z 113.464,A -85,B 0,C 180,E1 -13140,E2 -13140} C_VEL
LIN {X 0,Y 362.28,Z 113.485,A -85,B 0,C 180,E1 -13142.224,E2 -13142.224} C_VEL
LIN {X 0,Y 362.138,Z 113.498,A -85,B 0,C 180,E1 -13146.687,E2 -13146.687} C_VEL
LIN {X 0,Y 362.03,Z 113.515,A -85,B 0,C 180,E1 -13150.062,E2 -13150.062} C_VEL
LIN {X 0,Y 361.997,Z 113.52,A -85,B 0,C 180,E1 -13153.899,E2 -13153.899} C_VEL
LIN {X 0,Y 361.967,Z 113.522,A -85,B 0,C 180,E1 -13157.939,E2 -13157.939} C_VEL
LIN {X 0,Y 361.893,Z 113.533,A -85,B 0,C 180,E1 -13161.653,E2 -13161.653} C_VEL
LIN {X 0,Y 361.928,Z 113.527,A -85,B 0,C 180,E1 -13165.29,E2 -13165.29} C_VEL
LIN {X 0,Y 361.908,Z 113.528,A -85,B 0,C 180,E1 -13167.779,E2 -13167.779} C_VEL
LIN {X 0,Y 361.837,Z 113.537,A -85,B 0,C 180,E1 -13171.63,E2 -13171.63} C_VEL
LIN {X 0,Y 361.874,Z 113.534,A -85,B 0,C 180,E1 -13175.345,E2 -13175.345} C_VEL
LIN {X 0,Y 361.869,Z 113.537,A -85,B 0,C 180,E1 -13179.027,E2 -13179.027} C_VEL
LIN {X 0,Y 361.836,Z 113.54,A -85,B 0,C 180,E1 -13182.829,E2 -13182.829} C_VEL
LIN {X 0,Y 361.82,Z 113.537,A -85,B 0,C 180,E1 -13185.947,E2 -13185.947} C_VEL
LIN {X 0,Y 361.834,Z 113.536,A -85,B 0,C 180,E1 -13189.245,E2 -13189.245} C_VEL
LIN {X 0,Y 361.863,Z 113.536,A -85,B 0,C 180,E1 -13192.778,E2 -13192.778} C_VEL
LIN {X 0,Y 361.855,Z 113.533,A -85,B 0,C 180,E1 -13195.72,E2 -13195.72} C_VEL
LIN {X 0,Y 361.866,Z 113.532,A -85,B 0,C 180,E1 -13199.672,E2 -13199.672} C_VEL
LIN {X 0,Y 361.869,Z 113.531,A -85,B 0,C 180,E1 -13203.469,E2 -13203.469} C_VEL
LIN {X 0,Y 361.903,Z 113.629,A -85,B 0,C 180,E1 -13207.108,E2 -13207.108} C_VEL
LIN {X 0,Y 364.331,Z 124.588,A -85,B 0,C 180,E1 -13209.938,E2 -13209.938} C_VEL
LIN {X 0,Y 370.909,Z 142.142,A -85,B 0,C 180,E1 -13210.751,E2 -13210.751} C_VEL
LIN {X 0,Y 373.37,Z 154.733,A -85,B 0,C 180,E1 -13211.171,E2 -13211.171} C_VEL
